LIN {X 0,Y 573.073,Z 538.954,A -85,B 0,C 180,E1 -2243.185,E2 -2243.185} C_VEL
LIN {X 0,Y 573.07,Z 545.679,A -85,B 0,C 180,E1 -2244.369,E2 -2244.369} C_VEL
LIN {X 0,Y 573.028,Z 550.371,A -85,B 0,C 180,E1 -2245.427,E2 -2245.427} C_VEL
LIN {X 0,Y 573.022,Z 553.957,A -85,B 0,C 180,E1 -2246.484,E2 -2246.484} C_VEL
LIN {X 0,Y 572.959,Z 555.808,A -85,B 0,C 180,E1 -2247.187,E2 -2247.187} C_VEL
LIN {X 0,Y 572.939,Z 557.197,A -85,B 0,C 180,E1 -2247.891,E2 -2247.891} C_VEL
LIN {X 0,Y 572.941,Z 558.785,A -85,B 0,C 180,E1 -2249.297,E2 -2249.297} C_VEL
LIN {X 0,Y 572.938,Z 559,A -85,B 0,C 180,E1 -2250,E2 -2250} C_VEL
LIN {X 0,Y 572.946,Z 558.187,A -85,B 0,C 180,E1 -2251.405,E2 -2251.405} C_VEL
LIN {X 0,Y 572.939,Z 557.2,A -85,B 0,C 180,E1 -2252.109,E2 -2252.109} C_VEL
LIN {X 0,Y 572.959,Z 555.811,A -85,B 0,C 180,E1 -2252.812,E2 -2252.812} C_VEL
LIN {X 0,Y 573.014,Z 552.897,A -85,B 0,C 180,E1 -2253.868,E2 -2253.868} C_VEL
LIN {X 0,Y 572.963,Z 548.951,A -85,B 0,C 180,E1 -2254.925,E2 -2254.925} C_VEL
LIN {X 0,Y 573.064,Z 542.879,A -85,B 0,C 180,E1 -2256.16,E2 -2256.16} C_VEL
LIN {X 0,Y 573.119,Z 536.24,A -85,B 0,C 180,E1 -2257.22,E2 -2257.22} C_VEL
LIN {X 0,Y 573.2,Z 527.995,A -85,B 0,C 180,E1 -2258.283,E2 -2258.283} C_VEL
LIN {X 0,Y 573.286,Z 519.544,A -85,B 0,C 180,E1 -2259.17,E2 -2259.17} C_VEL
LIN {X 0,Y 573.43,Z 509.105,A -85,B 0,C 180,E1 -2260.058,E2 -2260.058} C_VEL
LIN {X 0,Y 573.549,Z 497.36,A -85,B 0,C 180,E1 -2260.857,E2 -2260.857} C_VEL
LIN {X 0,Y 573.652,Z 486.295,A -85,B 0,C 180,E1 -2261.447,E2 -2261.447} C_VEL
LIN {X 0,Y 573.758,Z 473.188,A -85,B 0,C 180,E1 -2261.973,E2 -2261.973} C_VEL
LIN {X 0,Y 573.831,Z 460.542,A -85,B 0,C 180,E1 -2262.331,E2 -2262.331} C_VEL
LIN {X 0,Y 573.923,Z 447.356,A -85,B 0,C 180,E1 -2262.553,E2 -2262.553} C_VEL
LIN {X 0,Y 574.016,Z 348.98,A -85,B 0,C 180,E1 -2263.79,E2 -2263.79} C_VEL
LIN {X 0,Y 573.511,Z 345.166,A -85,B 0,C 180,E1 -2263.87,E2 -2263.87} C_VEL
LIN {X 0,Y 573.751,Z 319.651,A -85,B 0,C 180,E1 -2266.729,E2 -2266.729} C_VEL
LIN {X 0,Y 574.013,Z 295.575,A -85,B 0,C 180,E1 -2269.479,E2 -2269.479} C_VEL
LIN {X 0,Y 574.248,Z 274.356,A -85,B 0,C 180,E1 -2271.917,E2 -2271.917} C_VEL
LIN {X 0,Y 574.374,Z 250.622,A -85,B 0,C 180,E1 -2274.583,E2 -2274.583} C_VEL
LIN {X 0,Y 574.422,Z 240.449,A -85,B 0,C 180,E1 -2275.742,E2 -2275.742} C_VEL
LIN {X 0,Y 573.225,Z 234.224,A -85,B 0,C 180,E1 -2276.525,E2 -2276.525} C_VEL
LIN {X 0,Y 573.208,Z 234.087,A -85,B 0,C 180,E1 -2279.368,E2 -2279.368} C_VEL
LIN {X 0,Y 573.223,Z 234.078,A -85,B 0,C 180,E1 -2282.223,E2 -2282.223} C_VEL
LIN {X 0,Y 573.207,Z 234.08,A -85,B 0,C 180,E1 -2284.767,E2 -2284.767} C_VEL
LIN {X 0,Y 573.181,Z 234.084,A -85,B 0,C 180,E1 -2287.81,E2 -2287.81} C_VEL
LIN {X 0,Y 573.201,Z 234.079,A -85,B 0,C 180,E1 -2290.527,E2 -2290.527} C_VEL
LIN {X 0,Y 573.184,Z 234.09,A -85,B 0,C 180,E1 -2293.363,E2 -2293.363} C_VEL
LIN {X 0,Y 573.192,Z 234.08,A -85,B 0,C 180,E1 -2296.335,E2 -2296.335} C_VEL
LIN {X 0,Y 573.236,Z 234.08,A -85,B 0,C 180,E1 -2299.474,E2 -2299.474} C_VEL
LIN {X 0,Y 573.203,Z 234.078,A -85,B 0,C 180,E1 -2302.19,E2 -2302.19} C_VEL
LIN {X 0,Y 573.21,Z 234.085,A -85,B 0,C 180,E1 -2305.23,E2 -2305.23} C_VEL
LIN {X 0,Y 573.205,Z 234.078,A -85,B 0,C 180,E1 -2308.182,E2 -2308.182} C_VEL
LIN {X 0,Y 573.212,Z 234.082,A -85,B 0,C 180,E1 -2310.631,E2 -2310.631} C_VEL
LIN {X 0,Y 573.188,Z 234.082,A -85,B 0,C 180,E1 -2313.514,E2 -2313.514} C_VEL
LIN {X 0,Y 573.178,Z 234.082,A -85,B 0,C 180,E1 -2316.132,E2 -2316.132} C_VEL
LIN {X 0,Y 573.22,Z 234.084,A -85,B 0,C 180,E1 -2318.713,E2 -2318.713} C_VEL
LIN {X 0,Y 573.18,Z 234.083,A -85,B 0,C 180,E1 -2321.41,E2 -2321.41} C_VEL
LIN {X 0,Y 573.2,Z 234.079,A -85,B 0,C 180,E1 -2323.62,E2 -2323.62} C_VEL
LIN {X 0,Y 573.211,Z 234.078,A -85,B 0,C 180,E1 -2325.806,E2 -2325.806} C_VEL
LIN {X 0,Y 573.248,Z 234.082,A -85,B 0,C 180,E1 -2328.745,E2 -2328.745} C_VEL
LIN {X 0,Y 573.214,Z 234.077,A -85,B 0,C 180,E1 -2331.54,E2 -2331.54} C_VEL
LIN {X 0,Y 573.258,Z 234.078,A -85,B 0,C 180,E1 -2334.372,E2 -2334.372} C_VEL
LIN {X 0,Y 573.265,Z 234.072,A -85,B 0,C 180,E1 -2337.189,E2 -2337.189} C_VEL
LIN {X 0,Y 573.283,Z 234.071,A -85,B 0,C 180,E1 -2340,E2 -2340} C_VEL
LIN {X 0,Y 573.276,Z 234.074,A -85,B 0,C 180,E1 -2342.811,E2 -2342.811} C_VEL
LIN {X 0,Y 573.242,Z 234.074,A -85,B 0,C 180,E1 -2345.629,E2 -2345.629} C_VEL
LIN {X 0,Y 573.22,Z 234.085,A -85,B 0,C 180,E1 -2348.461,E2 -2348.461} C_VEL
LIN {X 0,Y 573.22,Z 234.076,A -85,B 0,C 180,E1 -2351.313,E2 -2351.313} C_VEL
LIN {X 0,Y 573.249,Z 234.08,A -85,B 0,C 180,E1 -2354.417,E2 -2354.417} C_VEL
LIN {X 0,Y 573.203,Z 234.079,A -85,B 0,C 180,E1 -2357.114,E2 -2357.114} C_VEL
LIN {X 0,Y 573.215,Z 234.086,A -85,B 0,C 180,E1 -2360.078,E2 -2360.078} C_VEL
LIN {X 0,Y 573.223,Z 234.076,A -85,B 0,C 180,E1 -2363.1,E2 -2363.1} C_VEL
LIN {X 0,Y 573.2,Z 234.081,A -85,B 0,C 180,E1 -2364.386,E2 -2364.386} C_VEL
LIN {X 0,Y 572.558,Z 234.162,A -85,B 0,C 180,E1 -2364.973,E2 -2364.973} C_VEL
LIN {X 0,Y 569.714,Z 234.521,A -85,B 0,C 180,E1 -2365.924,E2 -2365.924} C_VEL
LIN {X 0,Y 567.285,Z 234.819,A -85,B 0,C 180,E1 -2366.69,E2 -2366.69} C_VEL
LIN {X 0,Y 566.226,Z 234.948,A -85,B 0,C 180,E1 -2367.281,E2 -2367.281} C_VEL
LIN {X 0,Y 566.133,Z 234.96,A -85,B 0,C 180,E1 -2367.481,E2 -2367.481} C_VEL
LIN {X 0,Y 566.154,Z 234.958,A -85,B 0,C 180,E1 -2370.595,E2 -2370.595} C_VEL
LIN {X 0,Y 566.151,Z 234.957,A -85,B 0,C 180,E1 -2373.107,E2 -2373.107} C_VEL
LIN {X 0,Y 566.127,Z 234.966,A -85,B 0,C 180,E1 -2375.695,E2 -2375.695} C_VEL
LIN {X 0,Y 566.177,Z 234.955,A -85,B 0,C 180,E1 -2378.556,E2 -2378.556} C_VEL
LIN {X 0,Y 566.127,Z 234.961,A -85,B 0,C 180,E1 -2381.144,E2 -2381.144} C_VEL
LIN {X 0,Y 566.137,Z 234.964,A -85,B 0,C 180,E1 -2384.042,E2 -2384.042} C_VEL
LIN {X 0,Y 566.176,Z 234.955,A -85,B 0,C 180,E1 -2387.086,E2 -2387.086} C_VEL
LIN {X 0,Y 566.178,Z 234.955,A -85,B 0,C 180,E1 -2390.32,E2 -2390.32} C_VEL
LIN {X 0,Y 566.179,Z 234.954,A -85,B 0,C 180,E1 -2392.603,E2 -2392.603} C_VEL
LIN {X 0,Y 566.169,Z 234.958,A -85,B 0,C 180,E1 -2395.181,E2 -2395.181} C_VEL
LIN {X 0,Y 566.209,Z 234.957,A -85,B 0,C 180,E1 -2397.743,E2 -2397.743} C_VEL
LIN {X 0,Y 566.148,Z 234.96,A -85,B 0,C 180,E1 -2401.045,E2 -2401.045} C_VEL
LIN {X 0,Y 566.166,Z 234.965,A -85,B 0,C 180,E1 -2403.457,E2 -2403.457} C_VEL
LIN {X 0,Y 566.15,Z 234.957,A -85,B 0,C 180,E1 -2406.595,E2 -2406.595} C_VEL
LIN {X 0,Y 566.19,Z 234.955,A -85,B 0,C 180,E1 -2408.902,E2 -2408.902} C_VEL
LIN {X 0,Y 566.167,Z 234.962,A -85,B 0,C 180,E1 -2411.172,E2 -2411.172} C_VEL
LIN {X 0,Y 566.163,Z 234.964,A -85,B 0,C 180,E1 -2413.412,E2 -2413.412} C_VEL
LIN {X 0,Y 566.156,Z 234.956,A -85,B 0,C 180,E1 -2416.358,E2 -2416.358} C_VEL
LIN {X 0,Y 566.216,Z 234.958,A -85,B 0,C 180,E1 -2419.27,E2 -2419.27} C_VEL
LIN {X 0,Y 566.172,Z 234.958,A -85,B 0,C 180,E1 -2422.153,E2 -2422.153} C_VEL
LIN {X 0,Y 566.215,Z 235.144,A -85,B 0,C 180,E1 -2424.168,E2 -2424.168} C_VEL
LIN {X 0,Y 566.455,Z 236.257,A -85,B 0,C 180,E1 -2424.282,E2 -2424.282} C_VEL
LIN {X 0,Y 567.145,Z 238.419,A -85,B 0,C 180,E1 -2424.333,E2 -2424.333} C_VEL
LIN {X 0,Y 566.959,Z 324.827,A -85,B 0,C 180,E1 -2425.446,E2 -2425.446} C_VEL
LIN {X 0,Y 566.876,Z 337.961,A -85,B 0,C 180,E1 -2425.757,E2 -2425.757} C_VEL
LIN {X 0,Y 566.752,Z 351.118,A -85,B 0,C 180,E1 -2426.223,E2 -2426.223} C_VEL
LIN {X 0,Y 566.582,Z 362.999,A -85,B 0,C 180,E1 -2426.801,E2 -2426.801} C_VEL
LIN {X 0,Y 566.441,Z 374.363,A -85,B 0,C 180,E1 -2427.511,E2 -2427.511} C_VEL
LIN {X 0,Y 566.31,Z 384.618,A -85,B 0,C 180,E1 -2428.311,E2 -2428.311} C_VEL
LIN {X 0,Y 566.199,Z 393.038,A -85,B 0,C 180,E1 -2429.111,E2 -2429.111} C_VEL
LIN {X 0,Y 566.093,Z 402.198,A -85,B 0,C 180,E1 -2430.178,E2 -2430.178} C_VEL
LIN {X 0,Y 566.004,Z 409.581,A -85,B 0,C 180,E1 -2431.245,E2 -2431.245} C_VEL
LIN {X 0,Y 565.957,Z 416.415,A -85,B 0,C 180,E1 -2432.491,E2 -2432.491} C_VEL
LIN {X 0,Y 565.953,Z 420.936,A -85,B 0,C 180,E1 -2433.56,E2 -2433.56} C_VEL
LIN {X 0,Y 565.937,Z 423.327,A -85,B 0,C 180,E1 -2434.273,E2 -2434.273} C_VEL
LIN {X 0,Y 565.854,Z 425.295,A -85,B 0,C 180,E1 -2434.988,E2 -2434.988} C_VEL
LIN {X 0,Y 565.905,Z 426.843,A -85,B 0,C 180,E1 -2435.702,E2 -2435.702} C_VEL
LIN {X 0,Y 565.921,Z 428.087,A -85,B 0,C 180,E1 -2436.534,E2 -2436.534} C_VEL
LIN {X 0,Y 565.879,Z 428.964,A -85,B 0,C 180,E1 -2437.852,E2 -2437.852} C_VEL
LIN {X 0,Y 565.853,Z 428.888,A -85,B 0,C 180,E1 -2438.572,E2 -2438.572} C_VEL
LIN {X 0,Y 565.829,Z 428.378,A -85,B 0,C 180,E1 -2439.292,E2 -2439.292} C_VEL
LIN {X 0,Y 565.883,Z 427.458,A -85,B 0,C 180,E1 -2440.013,E2 -2440.013} C_VEL
LIN {X 0,Y 565.905,Z 425.164,A -85,B 0,C 180,E1 -2441.153,E2 -2441.153} C_VEL
LIN {X 0,Y 565.926,Z 422.132,A -85,B 0,C 180,E1 -2442.188,E2 -2442.188} C_VEL
LIN {X 0,Y 565.938,Z 417.851,A -85,B 0,C 180,E1 -2443.282,E2 -2443.282} C_VEL
LIN {X 0,Y 565.966,Z 412.226,A -85,B 0,C 180,E1 -2444.398,E2 -2444.398} C_VEL
LIN {X 0,Y 566.052,Z 405.369,A -85,B 0,C 180,E1 -2445.482,E2 -2445.482} C_VEL
LIN {X 0,Y 566.145,Z 398.22,A -85,B 0,C 180,E1 -2446.404,E2 -2446.404} C_VEL
LIN {X 0,Y 566.271,Z 388.548,A -85,B 0,C 180,E1 -2447.422,E2 -2447.422} C_VEL
LIN {X 0,Y 566.386,Z 377.497,A -85,B 0,C 180,E1 -2448.353,E2 -2448.353} C_VEL
LIN {X 0,Y 566.562,Z 366.716,A -85,B 0,C 180,E1 -2449.077,E2 -2449.077} C_VEL
LIN {X 0,Y 566.696,Z 354.767,A -85,B 0,C 180,E1 -2449.704,E2 -2449.704} C_VEL
LIN {X 0,Y 566.847,Z 341.702,A -85,B 0,C 180,E1 -2450.219,E2 -2450.219} C_VEL
LIN {X 0,Y 566.948,Z 329.752,A -85,B 0,C 180,E1 -2450.546,E2 -2450.546} C_VEL
LIN {X 0,Y 566.981,Z 315.181,A -85,B 0,C 180,E1 -2450.782,E2 -2450.782} C_VEL
LIN {X 0,Y 567.039,Z 237.986,A -85,B 0,C 180,E1 -2451.765,E2 -2451.765} C_VEL
LIN {X 0,Y 566.316,Z 235.664,A -85,B 0,C 180,E1 -2451.847,E2 -2451.847} C_VEL
LIN {X 0,Y 566.185,Z 234.985,A -85,B 0,C 180,E1 -2452.006,E2 -2452.006} C_VEL
LIN {X 0,Y 566.181,Z 234.962,A -85,B 0,C 180,E1 -2455.021,E2 -2455.021} C_VEL
LIN {X 0,Y 566.167,Z 234.959,A -85,B 0,C 180,E1 -2457.341,E2 -2457.341} C_VEL
LIN {X 0,Y 566.17,Z 234.955,A -85,B 0,C 180,E1 -2459.77,E2 -2459.77} C_VEL
LIN {X 0,Y 566.202,Z 234.953,A -85,B 0,C 180,E1 -2462.429,E2 -2462.429} C_VEL
LIN {X 0,Y 566.17,Z 234.957,A -85,B 0,C 180,E1 -2464.987,E2 -2464.987} C_VEL
LIN {X 0,Y 566.184,Z 234.95,A -85,B 0,C 180,E1 -2467.461,E2 -2467.461} C_VEL
LIN {X 0,Y 566.204,Z 234.955,A -85,B 0,C 180,E1 -2470.199,E2 -2470.199} C_VEL
LIN {X 0,Y 566.185,Z 234.956,A -85,B 0,C 180,E1 -2473.055,E2 -2473.055} C_VEL
LIN {X 0,Y 566.153,Z 234.96,A -85,B 0,C 180,E1 -2476.053,E2 -2476.053} C_VEL
LIN {X 0,Y 566.198,Z 234.952,A -85,B 0,C 180,E1 -2479.214,E2 -2479.214} C_VEL
LIN {X 0,Y 566.171,Z 234.954,A -85,B 0,C 180,E1 -2481.635,E2 -2481.635} C_VEL
LIN {X 0,Y 566.138,Z 234.966,A -85,B 0,C 180,E1 -2484.306,E2 -2484.306} C_VEL
LIN {X 0,Y 566.204,Z 234.952,A -85,B 0,C 180,E1 -2486.896,E2 -2486.896} C_VEL
LIN {X 0,Y 566.169,Z 234.951,A -85,B 0,C 180,E1 -2489.406,E2 -2489.406} C_VEL
LIN {X 0,Y 566.164,Z 234.958,A -85,B 0,C 180,E1 -2491.854,E2 -2491.854} C_VEL
LIN {X 0,Y 566.231,Z 234.947,A -85,B 0,C 180,E1 -2495.038,E2 -2495.038} C_VEL
LIN {X 0,Y 566.178,Z 234.956,A -85,B 0,C 180,E1 -2498.136,E2 -2498.136} C_VEL
LIN {X 0,Y 566.223,Z 234.949,A -85,B 0,C 180,E1 -2500.613,E2 -2500.613} C_VEL
LIN {X 0,Y 566.169,Z 234.957,A -85,B 0,C 180,E1 -2503.411,E2 -2503.411} C_VEL
LIN {X 0,Y 566.172,Z 234.958,A -85,B 0,C 180,E1 -2506.358,E2 -2506.358} C_VEL
LIN {X 0,Y 566.222,Z 234.95,A -85,B 0,C 180,E1 -2509.27,E2 -2509.27} C_VEL
LIN {X 0,Y 566.18,Z 234.958,A -85,B 0,C 180,E1 -2512.152,E2 -2512.152} C_VEL
LIN {X 0,Y 566.256,Z 234.944,A -85,B 0,C 180,E1 -2515.016,E2 -2515.016} C_VEL
LIN {X 0,Y 566.259,Z 234.951,A -85,B 0,C 180,E1 -2517.866,E2 -2517.866} C_VEL
LIN {X 0,Y 566.267,Z 234.947,A -85,B 0,C 180,E1 -2520,E2 -2520} C_VEL
LIN {X 0,Y 566.241,Z 234.945,A -85,B 0,C 180,E1 -2522.846,E2 -2522.846} C_VEL
LIN {X 0,Y 566.231,Z 234.954,A -85,B 0,C 180,E1 -2525.698,E2 -2525.698} C_VEL
LIN {X 0,Y 566.178,Z 234.953,A -85,B 0,C 180,E1 -2528.566,E2 -2528.566} C_VEL
LIN {X 0,Y 566.23,Z 234.956,A -85,B 0,C 180,E1 -2531.454,E2 -2531.454} C_VEL
LIN {X 0,Y 566.193,Z 234.952,A -85,B 0,C 180,E1 -2534.494,E2 -2534.494} C_VEL
LIN {X 0,Y 566.177,Z 234.963,A -85,B 0,C 180,E1 -2537.332,E2 -2537.332} C_VEL
LIN {X 0,Y 566.189,Z 234.958,A -85,B 0,C 180,E1 -2539.581,E2 -2539.581} C_VEL
LIN {X 0,Y 566.174,Z 234.955,A -85,B 0,C 180,E1 -2541.863,E2 -2541.863} C_VEL
LIN {X 0,Y 566.17,Z 234.962,A -85,B 0,C 180,E1 -2545.021,E2 -2545.021} C_VEL
LIN {X 0,Y 566.154,Z 234.961,A -85,B 0,C 180,E1 -2547.342,E2 -2547.342} C_VEL
LIN {X 0,Y 566.15,Z 234.959,A -85,B 0,C 180,E1 -2549.772,E2 -2549.772} C_VEL
LIN {X 0,Y 566.183,Z 234.954,A -85,B 0,C 180,E1 -2552.428,E2 -2552.428} C_VEL
LIN {X 0,Y 566.158,Z 234.964,A -85,B 0,C 180,E1 -2554.988,E2 -2554.988} C_VEL
LIN {X 0,Y 566.178,Z 234.956,A -85,B 0,C 180,E1 -2557.462,E2 -2557.462} C_VEL
LIN {X 0,Y 566.199,Z 234.952,A -85,B 0,C 180,E1 -2560.2,E2 -2560.2} C_VEL
LIN {X 0,Y 566.141,Z 234.964,A -85,B 0,C 180,E1 -2563.06,E2 -2563.06} C_VEL
LIN {X 0,Y 566.14,Z 234.959,A -85,B 0,C 180,E1 -2566.055,E2 -2566.055} C_VEL
LIN {X 0,Y 566.141,Z 234.965,A -85,B 0,C 180,E1 -2568.858,E2 -2568.858} C_VEL
LIN {X 0,Y 566.153,Z 234.957,A -85,B 0,C 180,E1 -2571.45,E2 -2571.45} C_VEL
LIN {X 0,Y 566.151,Z 234.958,A -85,B 0,C 180,E1 -2573.793,E2 -2573.793} C_VEL
LIN {X 0,Y 566.193,Z 234.957,A -85,B 0,C 180,E1 -2576.269,E2 -2576.269} C_VEL
LIN {X 0,Y 566.166,Z 234.961,A -85,B 0,C 180,E1 -2578.928,E2 -2578.928} C_VEL
LIN {X 0,Y 566.134,Z 234.964,A -85,B 0,C 180,E1 -2581.854,E2 -2581.854} C_VEL
LIN {X 0,Y 566.18,Z 235.187,A -85,B 0,C 180,E1 -2583.372,E2 -2583.372} C_VEL
LIN {X 0,Y 567.401,Z 241.103,A -85,B 0,C 180,E1 -2584.112,E2 -2584.112} C_VEL
LIN {X 0,Y 567.362,Z 259.698,A -85,B 0,C 180,E1 -2586.243,E2 -2586.243} C_VEL
LIN {X 0,Y 567.226,Z 283.598,A -85,B 0,C 180,E1 -2588.942,E2 -2588.942} C_VEL
LIN {X 0,Y 566.989,Z 303.539,A -85,B 0,C 180,E1 -2591.199,E2 -2591.199} C_VEL
LIN {X 0,Y 566.733,Z 326.088,A -85,B 0,C 180,E1 -2593.798,E2 -2593.798} C_VEL
LIN {X 0,Y 566.548,Z 345.155,A -85,B 0,C 180,E1 -2595.956,E2 -2595.956} C_VEL
LIN {X 0,Y 567.173,Z 350.721,A -85,B 0,C 180,E1 -2596.063,E2 -2596.063} C_VEL
LIN {X 0,Y 566.975,Z 454.945,A -85,B 0,C 180,E1 -2597.403,E2 -2597.403} C_VEL
LIN {X 0,Y 566.867,Z 468.217,A -85,B 0,C 180,E1 -2597.719,E2 -2597.719} C_VEL
LIN {X 0,Y 566.728,Z 481.153,A -85,B 0,C 180,E1 -2598.179,E2 -2598.179} C_VEL
LIN {X 0,Y 566.604,Z 493.246,A -85,B 0,C 180,E1 -2598.77,E2 -2598.77} C_VEL
LIN {X 0,Y 566.425,Z 505.483,A -85,B 0,C 180,E1 -2599.545,E2 -2599.545} C_VEL
LIN {X 0,Y 566.297,Z 515.646,A -85,B 0,C 180,E1 -2600.355,E2 -2600.355} C_VEL
LIN {X 0,Y 566.166,Z 524.785,A -85,B 0,C 180,E1 -2601.253,E2 -2601.253} C_VEL
LIN {X 0,Y 566.081,Z 533.688,A -85,B 0,C 180,E1 -2602.33,E2 -2602.33} C_VEL
LIN {X 0,Y 565.967,Z 540.955,A -85,B 0,C 180,E1 -2603.422,E2 -2603.422} C_VEL
LIN {X 0,Y 566.004,Z 545.679,A -85,B 0,C 180,E1 -2604.299,E2 -2604.299} C_VEL
LIN {X 0,Y 565.933,Z 550.372,A -85,B 0,C 180,E1 -2605.37,E2 -2605.37} C_VEL
LIN {X 0,Y 565.927,Z 553.957,A -85,B 0,C 180,E1 -2606.44,E2 -2606.44} C_VEL
LIN {X 0,Y 565.878,Z 555.807,A -85,B 0,C 180,E1 -2607.152,E2 -2607.152} C_VEL
LIN {X 0,Y 565.846,Z 558.184,A -85,B 0,C 180,E1 -2608.576,E2 -2608.576} C_VEL
LIN {X 0,Y 565.839,Z 559,A -85,B 0,C 180,E1 -2610,E2 -2610} C_VEL
LIN {X 0,Y 565.846,Z 558.186,A -85,B 0,C 180,E1 -2611.423,E2 -2611.423} C_VEL
LIN {X 0,Y 565.878,Z 555.811,A -85,B 0,C 180,E1 -2612.847,E2 -2612.847} C_VEL
LIN {X 0,Y 565.926,Z 552.897,A -85,B 0,C 180,E1 -2613.916,E2 -2613.916} C_VEL
LIN {X 0,Y 565.878,Z 548.95,A -85,B 0,C 180,E1 -2614.987,E2 -2614.987} C_VEL
LIN {X 0,Y 566.002,Z 543.869,A -85,B 0,C 180,E1 -2616.058,E2 -2616.058} C_VEL
LIN {X 0,Y 566.039,Z 537.471,A -85,B 0,C 180,E1 -2617.132,E2 -2617.132} C_VEL
LIN {X 0,Y 566.133,Z 529.482,A -85,B 0,C 180,E1 -2618.207,E2 -2618.207} C_VEL
LIN {X 0,Y 566.228,Z 521.34,A -85,B 0,C 180,E1 -2619.105,E2 -2619.105} C_VEL
LIN {X 0,Y 566.35,Z 511.406,A -85,B 0,C 180,E1 -2620.004,E2 -2620.004} C_VEL
LIN {X 0,Y 566.525,Z 500.294,A -85,B 0,C 180,E1 -2620.807,E2 -2620.807} C_VEL
LIN {X 0,Y 566.659,Z 489.186,A -85,B 0,C 180,E1 -2621.445,E2 -2621.445} C_VEL
LIN {X 0,Y 566.741,Z 476.996,A -85,B 0,C 180,E1 -2621.988,E2 -2621.988} C_VEL
LIN {X 0,Y 566.886,Z 464.199,A -85,B 0,C 180,E1 -2622.393,E2 -2622.393} C_VEL
LIN {X 0,Y 566.964,Z 450.64,A -85,B 0,C 180,E1 -2622.664,E2 -2622.664} C_VEL
LIN {X 0,Y 567.122,Z 349.652,A -85,B 0,C 180,E1 -2623.952,E2 -2623.952} C_VEL
LIN {X 0,Y 566.559,Z 345.174,A -85,B 0,C 180,E1 -2624.043,E2 -2624.043} C_VEL
LIN {X 0,Y 566.814,Z 319.831,A -85,B 0,C 180,E1 -2626.919,E2 -2626.919} C_VEL
LIN {X 0,Y 567.118,Z 295.582,A -85,B 0,C 180,E1 -2629.717,E2 -2629.717} C_VEL
LIN {X 0,Y 567.331,Z 270.088,A -85,B 0,C 180,E1 -2632.582,E2 -2632.582} C_VEL
LIN {X 0,Y 567.506,Z 243.009,A -85,B 0,C 180,E1 -2635.685,E2 -2635.685} C_VEL
LIN {X 0,Y 566.731,Z 237.816,A -85,B 0,C 180,E1 -2636.316,E2 -2636.316} C_VEL
LIN {X 0,Y 566.178,Z 235.079,A -85,B 0,C 180,E1 -2636.689,E2 -2636.689} C_VEL
LIN {X 0,Y 566.141,Z 234.966,A -85,B 0,C 180,E1 -2639.771,E2 -2639.771} C_VEL
LIN {X 0,Y 566.171,Z 234.956,A -85,B 0,C 180,E1 -2642.424,E2 -2642.424} C_VEL
LIN {X 0,Y 566.152,Z 234.961,A -85,B 0,C 180,E1 -2644.985,E2 -2644.985} C_VEL
LIN {X 0,Y 566.17,Z 234.963,A -85,B 0,C 180,E1 -2647.462,E2 -2647.462} C_VEL
LIN {X 0,Y 566.154,Z 234.957,A -85,B 0,C 180,E1 -2650.202,E2 -2650.202} C_VEL
LIN {X 0,Y 566.135,Z 234.965,A -85,B 0,C 180,E1 -2653.059,E2 -2653.059} C_VEL
LIN {X 0,Y 566.143,Z 234.958,A -85,B 0,C 180,E1 -2656.053,E2 -2656.053} C_VEL
LIN {X 0,Y 566.162,Z 234.965,A -85,B 0,C 180,E1 -2659.218,E2 -2659.218} C_VEL
LIN {X 0,Y 566.16,Z 234.959,A -85,B 0,C 180,E1 -2661.635,E2 -2661.635} C_VEL
LIN {X 0,Y 566.126,Z 234.961,A -85,B 0,C 180,E1 -2664.305,E2 -2664.305} C_VEL
LIN {X 0,Y 566.149,Z 234.965,A -85,B 0,C 180,E1 -2666.893,E2 -2666.893} C_VEL
LIN {X 0,Y 566.145,Z 234.962,A -85,B 0,C 180,E1 -2669.405,E2 -2669.405} C_VEL
LIN {X 0,Y 566.134,Z 234.959,A -85,B 0,C 180,E1 -2671.853,E2 -2671.853} C_VEL
LIN {X 0,Y 566.161,Z 234.957,A -85,B 0,C 180,E1 -2674.248,E2 -2674.248} C_VEL
LIN {X 0,Y 566.144,Z 234.961,A -85,B 0,C 180,E1 -2677.367,E2 -2677.367} C_VEL
LIN {X 0,Y 566.155,Z 234.957,A -85,B 0,C 180,E1 -2679.661,E2 -2679.661} C_VEL
LIN {X 0,Y 566.154,Z 234.957,A -85,B 0,C 180,E1 -2681.92,E2 -2681.92} C_VEL
LIN {X 0,Y 566.165,Z 234.963,A -85,B 0,C 180,E1 -2684.89,E2 -2684.89} C_VEL
LIN {X 0,Y 566.16,Z 234.956,A -85,B 0,C 180,E1 -2687.817,E2 -2687.817} C_VEL
LIN {X 0,Y 566.136,Z 234.96,A -85,B 0,C 180,E1 -2689.992,E2 -2689.992} C_VEL
LIN {X 0,Y 566.195,Z 234.958,A -85,B 0,C 180,E1 -2692.87,E2 -2692.87} C_VEL
LIN {X 0,Y 566.24,Z 234.949,A -85,B 0,C 180,E1 -2695.016,E2 -2695.016} C_VEL
LIN {X 0,Y 566.242,Z 234.947,A -85,B 0,C 180,E1 -2697.866,E2 -2697.866} C_VEL
LIN {X 0,Y 566.283,Z 234.947,A -85,B 0,C 180,E1 -2700.711,E2 -2700.711} C_VEL
LIN {X 0,Y 566.24,Z 234.95,A -85,B 0,C 180,E1 -2702.846,E2 -2702.846} C_VEL
LIN {X 0,Y 566.212,Z 234.95,A -85,B 0,C 180,E1 -2705.699,E2 -2705.699} C_VEL
LIN {X 0,Y 566.173,Z 234.961,A -85,B 0,C 180,E1 -2708.567,E2 -2708.567} C_VEL
LIN {X 0,Y 566.178,Z 234.954,A -85,B 0,C 180,E1 -2711.456,E2 -2711.456} C_VEL
LIN {X 0,Y 566.204,Z 234.957,A -85,B 0,C 180,E1 -2714.5,E2 -2714.5} C_VEL
LIN {X 0,Y 566.156,Z 234.957,A -85,B 0,C 180,E1 -2717.333,E2 -2717.333} C_VEL
LIN {X 0,Y 566.184,Z 234.955,A -85,B 0,C 180,E1 -2719.582,E2 -2719.582} C_VEL
LIN {X 0,Y 566.169,Z 234.96,A -85,B 0,C 180,E1 -2721.864,E2 -2721.864} C_VEL
LIN {X 0,Y 566.166,Z 234.955,A -85,B 0,C 180,E1 -2725.022,E2 -2725.022} C_VEL
LIN {X 0,Y 566.133,Z 234.96,A -85,B 0,C 180,E1 -2727.481,E2 -2727.481} C_VEL
LIN {X 0,Y 565.447,Z 235.054,A -85,B 0,C 180,E1 -2728.075,E2 -2728.075} C_VEL
LIN {X 0,Y 562.594,Z 235.407,A -85,B 0,C 180,E1 -2729.039,E2 -2729.039} C_VEL
LIN {X 0,Y 560.203,Z 235.705,A -85,B 0,C 180,E1 -2729.815,E2 -2729.815} C_VEL
LIN {X 0,Y 559.189,Z 235.828,A -85,B 0,C 180,E1 -2730.414,E2 -2730.414} C_VEL
LIN {X 0,Y 559.113,Z 235.835,A -85,B 0,C 180,E1 -2730.616,E2 -2730.616} C_VEL
LIN {X 0,Y 559.124,Z 235.833,A -85,B 0,C 180,E1 -2732.718,E2 -2732.718} C_VEL
LIN {X 0,Y 559.103,Z 235.837,A -85,B 0,C 180,E1 -2735.326,E2 -2735.326} C_VEL
LIN {X 0,Y 559.105,Z 235.842,A -85,B 0,C 180,E1 -2738.02,E2 -2738.02} C_VEL
LIN {X 0,Y 559.083,Z 235.838,A -85,B 0,C 180,E1 -2740.819,E2 -2740.819} C_VEL
LIN {X 0,Y 559.084,Z 235.847,A -85,B 0,C 180,E1 -2743.74,E2 -2743.74} C_VEL
LIN {X 0,Y 559.098,Z 235.838,A -85,B 0,C 180,E1 -2746.264,E2 -2746.264} C_VEL
LIN {X 0,Y 559.085,Z 235.84,A -85,B 0,C 180,E1 -2749.183,E2 -2749.183} C_VEL
LIN {X 0,Y 559.115,Z 235.838,A -85,B 0,C 180,E1 -2751.982,E2 -2751.982} C_VEL
LIN {X 0,Y 559.112,Z 235.834,A -85,B 0,C 180,E1 -2754.791,E2 -2754.791} C_VEL
LIN {X 0,Y 559.138,Z 235.837,A -85,B 0,C 180,E1 -2757.368,E2 -2757.368} C_VEL
LIN {X 0,Y 559.099,Z 235.837,A -85,B 0,C 180,E1 -2760.153,E2 -2760.153} C_VEL
LIN {X 0,Y 559.107,Z 235.84,A -85,B 0,C 180,E1 -2763.187,E2 -2763.187} C_VEL
LIN {X 0,Y 559.089,Z 235.846,A -85,B 0,C 180,E1 -2765.493,E2 -2765.493} C_VEL
LIN {X 0,Y 559.131,Z 235.832,A -85,B 0,C 180,E1 -2768.458,E2 -2768.458} C_VEL
LIN {X 0,Y 559.135,Z 235.835,A -85,B 0,C 180,E1 -2770.926,E2 -2770.926} C_VEL
LIN {X 0,Y 559.142,Z 235.838,A -85,B 0,C 180,E1 -2773.197,E2 -2773.197} C_VEL
LIN {X 0,Y 559.135,Z 235.831,A -85,B 0,C 180,E1 -2776.184,E2 -2776.184} C_VEL
LIN {X 0,Y 559.173,Z 235.836,A -85,B 0,C 180,E1 -2779.134,E2 -2779.134} C_VEL
LIN {X 0,Y 559.127,Z 235.836,A -85,B 0,C 180,E1 -2782.053,E2 -2782.053} C_VEL
LIN {X 0,Y 559.174,Z 236.047,A -85,B 0,C 180,E1 -2784.003,E2 -2784.003} C_VEL
LIN {X 0,Y 559.421,Z 237.127,A -85,B 0,C 180,E1 -2784.114,E2 -2784.114} C_VEL
LIN {X 0,Y 560.214,Z 239.499,A -85,B 0,C 180,E1 -2784.173,E2 -2784.173} C_VEL
LIN {X 0,Y 560.037,Z 325.412,A -85,B 0,C 180,E1 -2785.299,E2 -2785.299} C_VEL
LIN {X 0,Y 559.929,Z 339.105,A -85,B 0,C 180,E1 -2785.636,E2 -2785.636} C_VEL
LIN {X 0,Y 559.805,Z 351.403,A -85,B 0,C 180,E1 -2786.086,E2 -2786.086} C_VEL
LIN {X 0,Y 559.611,Z 363.203,A -85,B 0,C 180,E1 -2786.671,E2 -2786.671} C_VEL
LIN {X 0,Y 559.446,Z 374.53,A -85,B 0,C 180,E1 -2787.39,E2 -2787.39} C_VEL
LIN {X 0,Y 559.298,Z 384.759,A -85,B 0,C 180,E1 -2788.2,E2 -2788.2} C_VEL
LIN {X 0,Y 559.137,Z 394.002,A -85,B 0,C 180,E1 -2789.1,E2 -2789.1} C_VEL
LIN {X 0,Y 559.033,Z 402.96,A -85,B 0,C 180,E1 -2790.18,E2 -2790.18} C_VEL
LIN {X 0,Y 558.926,Z 410.21,A -85,B 0,C 180,E1 -2791.261,E2 -2791.261} C_VEL
LIN {X 0,Y 558.855,Z 416.876,A -85,B 0,C 180,E1 -2792.523,E2 -2792.523} C_VEL
LIN {X 0,Y 558.858,Z 421.29,A -85,B 0,C 180,E1 -2793.605,E2 -2793.605} C_VEL
LIN {X 0,Y 558.828,Z 423.63,A -85,B 0,C 180,E1 -2794.328,E2 -2794.328} C_VEL
LIN {X 0,Y 558.769,Z 425.547,A -85,B 0,C 180,E1 -2795.051,E2 -2795.051} C_VEL
LIN {X 0,Y 558.816,Z 427.029,A -85,B 0,C 180,E1 -2795.775,E2 -2795.775} C_VEL
LIN {X 0,Y 558.849,Z 428.109,A -85,B 0,C 180,E1 -2796.536,E2 -2796.536} C_VEL
LIN {X 0,Y 558.797,Z 428.986,A -85,B 0,C 180,E1 -2797.952,E2 -2797.952} C_VEL
LIN {X 0,Y 558.767,Z 428.84,A -85,B 0,C 180,E1 -2798.681,E2 -2798.681} C_VEL
LIN {X 0,Y 558.78,Z 427.295,A -85,B 0,C 180,E1 -2800.142,E2 -2800.142} C_VEL
LIN {X 0,Y 558.807,Z 425.177,A -85,B 0,C 180,E1 -2801.187,E2 -2801.187} C_VEL
LIN {X 0,Y 558.835,Z 421.772,A -85,B 0,C 180,E1 -2802.345,E2 -2802.345} C_VEL
LIN {X 0,Y 558.851,Z 417.383,A -85,B 0,C 180,E1 -2803.453,E2 -2803.453} C_VEL
LIN {X 0,Y 558.914,Z 411.744,A -85,B 0,C 180,E1 -2804.566,E2 -2804.566} C_VEL
LIN {X 0,Y 558.985,Z 404.643,A -85,B 0,C 180,E1 -2805.683,E2 -2805.683} C_VEL
LIN {X 0,Y 559.104,Z 397.338,A -85,B 0,C 180,E1 -2806.617,E2 -2806.617} C_VEL
LIN {X 0,Y 559.273,Z 387.405,A -85,B 0,C 180,E1 -2807.648,E2 -2807.648} C_VEL
LIN {X 0,Y 559.397,Z 377.334,A -85,B 0,C 180,E1 -2808.495,E2 -2808.495} C_VEL
LIN {X 0,Y 559.577,Z 366.85,A -85,B 0,C 180,E1 -2809.208,E2 -2809.208} C_VEL
LIN {X 0,Y 559.723,Z 354.486,A -85,B 0,C 180,E1 -2809.865,E2 -2809.865} C_VEL
LIN {X 0,Y 559.887,Z 342.693,A -85,B 0,C 180,E1 -2810.337,E2 -2810.337} C_VEL
LIN {X 0,Y 560.021,Z 330.255,A -85,B 0,C 180,E1 -2810.692,E2 -2810.692} C_VEL
LIN {X 0,Y 560.058,Z 316.069,A -85,B 0,C 180,E1 -2810.931,E2 -2810.931} C_VEL
LIN {X 0,Y 560.197,Z 239.496,A -85,B 0,C 180,E1 -2811.918,E2 -2811.918} C_VEL
LIN {X 0,Y 559.278,Z 236.553,A -85,B 0,C 180,E1 -2812.014,E2 -2812.014} C_VEL
LIN {X 0,Y 559.153,Z 235.877,A -85,B 0,C 180,E1 -2812.152,E2 -2812.152} C_VEL
LIN {X 0,Y 559.127,Z 235.838,A -85,B 0,C 180,E1 -2815.3,E2 -2815.3} C_VEL
LIN {X 0,Y 559.136,Z 235.835,A -85,B 0,C 180,E1 -2818.374,E2 -2818.374} C_VEL
LIN {X 0,Y 559.142,Z 235.831,A -85,B 0,C 180,E1 -2821.271,E2 -2821.271} C_VEL
LIN {X 0,Y 559.154,Z 235.831,A -85,B 0,C 180,E1 -2823.946,E2 -2823.946} C_VEL
LIN {X 0,Y 559.124,Z 235.832,A -85,B 0,C 180,E1 -2827.109,E2 -2827.109} C_VEL
LIN {X 0,Y 559.155,Z 235.831,A -85,B 0,C 180,E1 -2829.94,E2 -2829.94} C_VEL
LIN {X 0,Y 559.148,Z 235.837,A -85,B 0,C 180,E1 -2832.744,E2 -2832.744} C_VEL
LIN {X 0,Y 559.121,Z 235.834,A -85,B 0,C 180,E1 -2835.763,E2 -2835.763} C_VEL
LIN {X 0,Y 559.12,Z 235.837,A -85,B 0,C 180,E1 -2838.225,E2 -2838.225} C_VEL
LIN {X 0,Y 559.165,Z 235.826,A -85,B 0,C 180,E1 -2841.192,E2 -2841.192} C_VEL
LIN {X 0,Y 559.111,Z 235.834,A -85,B 0,C 180,E1 -2843.787,E2 -2843.787} C_VEL
LIN {X 0,Y 559.154,Z 235.836,A -85,B 0,C 180,E1 -2846.424,E2 -2846.424} C_VEL
LIN {X 0,Y 559.145,Z 235.826,A -85,B 0,C 180,E1 -2848.98,E2 -2848.98} C_VEL
LIN {X 0,Y 559.111,Z 235.834,A -85,B 0,C 180,E1 -2851.628,E2 -2851.628} C_VEL
LIN {X 0,Y 559.155,Z 235.83,A -85,B 0,C 180,E1 -2854.817,E2 -2854.817} C_VEL
LIN {X 0,Y 559.126,Z 235.833,A -85,B 0,C 180,E1 -2857.846,E2 -2857.846} C_VEL
LIN {X 0,Y 559.185,Z 235.827,A -85,B 0,C 180,E1 -2860.494,E2 -2860.494} C_VEL
LIN {X 0,Y 559.147,Z 235.83,A -85,B 0,C 180,E1 -2863.196,E2 -2863.196} C_VEL
LIN {X 0,Y 559.148,Z 235.835,A -85,B 0,C 180,E1 -2866.183,E2 -2866.183} C_VEL
LIN {X 0,Y 559.181,Z 235.826,A -85,B 0,C 180,E1 -2869.133,E2 -2869.133} C_VEL
LIN {X 0,Y 559.133,Z 235.837,A -85,B 0,C 180,E1 -2872.052,E2 -2872.052} C_VEL
LIN {X 0,Y 559.23,Z 235.819,A -85,B 0,C 180,E1 -2874.953,E2 -2874.953} C_VEL
LIN {X 0,Y 559.232,Z 235.827,A -85,B 0,C 180,E1 -2877.839,E2 -2877.839} C_VEL
LIN {X 0,Y 559.237,Z 235.822,A -85,B 0,C 180,E1 -2880,E2 -2880} C_VEL
LIN {X 0,Y 559.21,Z 235.821,A -85,B 0,C 180,E1 -2882.881,E2 -2882.881} C_VEL
LIN {X 0,Y 559.197,Z 235.829,A -85,B 0,C 180,E1 -2885.77,E2 -2885.77} C_VEL
LIN {X 0,Y 559.145,Z 235.829,A -85,B 0,C 180,E1 -2888.675,E2 -2888.675} C_VEL
LIN {X 0,Y 559.187,Z 235.831,A -85,B 0,C 180,E1 -2891.601,E2 -2891.601} C_VEL
LIN {X 0,Y 559.143,Z 235.83,A -85,B 0,C 180,E1 -2894.576,E2 -2894.576} C_VEL
LIN {X 0,Y 559.121,Z 235.838,A -85,B 0,C 180,E1 -2897.558,E2 -2897.558} C_VEL
LIN {X 0,Y 559.152,Z 235.831,A -85,B 0,C 180,E1 -2899.838,E2 -2899.838} C_VEL
LIN {X 0,Y 559.12,Z 235.832,A -85,B 0,C 180,E1 -2902.154,E2 -2902.154} C_VEL
LIN {X 0,Y 559.13,Z 235.841,A -85,B 0,C 180,E1 -2905.178,E2 -2905.178} C_VEL
LIN {X 0,Y 559.098,Z 235.835,A -85,B 0,C 180,E1 -2907.717,E2 -2907.717} C_VEL
LIN {X 0,Y 559.093,Z 235.837,A -85,B 0,C 180,E1 -2910.186,E2 -2910.186} C_VEL
LIN {X 0,Y 559.139,Z 235.835,A -85,B 0,C 180,E1 -2912.716,E2 -2912.716} C_VEL
LIN {X 0,Y 559.108,Z 235.839,A -85,B 0,C 180,E1 -2915.326,E2 -2915.326} C_VEL
LIN {X 0,Y 559.115,Z 235.833,A -85,B 0,C 180,E1 -2918.019,E2 -2918.019} C_VEL
LIN {X 0,Y 559.119,Z 235.842,A -85,B 0,C 180,E1 -2920.816,E2 -2920.816} C_VEL
LIN {X 0,Y 559.093,Z 235.836,A -85,B 0,C 180,E1 -2923.739,E2 -2923.739} C_VEL
LIN {X 0,Y 559.088,Z 235.84,A -85,B 0,C 180,E1 -2926.262,E2 -2926.262} C_VEL
LIN {X 0,Y 559.098,Z 235.837,A -85,B 0,C 180,E1 -2929.183,E2 -2929.183} C_VEL
LIN {X 0,Y 559.094,Z 235.837,A -85,B 0,C 180,E1 -2931.98,E2 -2931.98} C_VEL
LIN {X 0,Y 559.114,Z 235.839,A -85,B 0,C 180,E1 -2934.79,E2 -2934.79} C_VEL
LIN {X 0,Y 559.133,Z 235.832,A -85,B 0,C 180,E1 -2937.368,E2 -2937.368} C_VEL
LIN {X 0,Y 559.093,Z 235.843,A -85,B 0,C 180,E1 -2940.153,E2 -2940.153} C_VEL
LIN {X 0,Y 559.126,Z 235.932,A -85,B 0,C 180,E1 -2943.182,E2 -2943.182} C_VEL
LIN {X 0,Y 560.52,Z 243.305,A -85,B 0,C 180,E1 -2944.133,E2 -2944.133} C_VEL
LIN {X 0,Y 560.376,Z 267.452,A -85,B 0,C 180,E1 -2946.926,E2 -2946.926} C_VEL
LIN {X 0,Y 560.146,Z 292.823,A -85,B 0,C 180,E1 -2949.816,E2 -2949.816} C_VEL
LIN {X 0,Y 559.897,Z 318.228,A -85,B 0,C 180,E1 -2952.681,E2 -2952.681} C_VEL
LIN {X 0,Y 559.589,Z 344.862,A -85,B 0,C 180,E1 -2955.754,E2 -2955.754} C_VEL
LIN {X 0,Y 559.791,Z 347.143,A -85,B 0,C 180,E1 -2955.829,E2 -2955.829} C_VEL
LIN {X 0,Y 560.328,Z 352.509,A -85,B 0,C 180,E1 -2955.912,E2 -2955.912} C_VEL
LIN {X 0,Y 560.058,Z 454.945,A -85,B 0,C 180,E1 -2957.245,E2 -2957.245} C_VEL
LIN {X 0,Y 559.946,Z 468.217,A -85,B 0,C 180,E1 -2957.565,E2 -2957.565} C_VEL
LIN {X 0,Y 559.792,Z 481.155,A -85,B 0,C 180,E1 -2958.031,E2 -2958.031} C_VEL
LIN {X 0,Y 559.634,Z 493.845,A -85,B 0,C 180,E1 -2958.663,E2 -2958.663} C_VEL
LIN {X 0,Y 559.443,Z 505.485,A -85,B 0,C 180,E1 -2959.413,E2 -2959.413} C_VEL
LIN {X 0,Y 559.294,Z 515.646,A -85,B 0,C 180,E1 -2960.233,E2 -2960.233} C_VEL
LIN {X 0,Y 559.134,Z 524.785,A -85,B 0,C 180,E1 -2961.143,E2 -2961.143} C_VEL
LIN {X 0,Y 559.009,Z 533.688,A -85,B 0,C 180,E1 -2962.232,E2 -2962.232} C_VEL
LIN {X 0,Y 558.925,Z 539.739,A -85,B 0,C 180,E1 -2963.14,E2 -2963.14} C_VEL
LIN {X 0,Y 558.935,Z 545.679,A -85,B 0,C 180,E1 -2964.227,E2 -2964.227} C_VEL
LIN {X 0,Y 558.826,Z 550.372,A -85,B 0,C 180,E1 -2965.311,E2 -2965.311} C_VEL
LIN {X 0,Y 558.836,Z 553.957,A -85,B 0,C 180,E1 -2966.395,E2 -2966.395} C_VEL
LIN {X 0,Y 558.799,Z 555.807,A -85,B 0,C 180,E1 -2967.116,E2 -2967.116} C_VEL
LIN {X 0,Y 558.746,Z 558.184,A -85,B 0,C 180,E1 -2968.558,E2 -2968.558} C_VEL
LIN {X 0,Y 558.74,Z 559,A -85,B 0,C 180,E1 -2970,E2 -2970} C_VEL
LIN {X 0,Y 558.746,Z 558.185,A -85,B 0,C 180,E1 -2971.441,E2 -2971.441} C_VEL
LIN {X 0,Y 558.799,Z 555.811,A -85,B 0,C 180,E1 -2972.883,E2 -2972.883} C_VEL
LIN {X 0,Y 558.843,Z 552.897,A -85,B 0,C 180,E1 -2973.966,E2 -2973.966} C_VEL
LIN {X 0,Y 558.798,Z 548.95,A -85,B 0,C 180,E1 -2975.05,E2 -2975.05} C_VEL
LIN {X 0,Y 558.919,Z 543.869,A -85,B 0,C 180,E1 -2976.135,E2 -2976.135} C_VEL
LIN {X 0,Y 558.977,Z 537.471,A -85,B 0,C 180,E1 -2977.222,E2 -2977.222} C_VEL
LIN {X 0,Y 559.098,Z 529.482,A -85,B 0,C 180,E1 -2978.311,E2 -2978.311} C_VEL
LIN {X 0,Y 559.184,Z 521.339,A -85,B 0,C 180,E1 -2979.221,E2 -2979.221} C_VEL
LIN {X 0,Y 559.359,Z 511.405,A -85,B 0,C 180,E1 -2980.131,E2 -2980.131} C_VEL
LIN {X 0,Y 559.53,Z 500.373,A -85,B 0,C 180,E1 -2980.939,E2 -2980.939} C_VEL
LIN {X 0,Y 559.702,Z 488.151,A -85,B 0,C 180,E1 -2981.643,E2 -2981.643} C_VEL
LIN {X 0,Y 559.83,Z 475.784,A -85,B 0,C 180,E1 -2982.184,E2 -2982.184} C_VEL
LIN {X 0,Y 559.983,Z 462.369,A -85,B 0,C 180,E1 -2982.595,E2 -2982.595} C_VEL
LIN {X 0,Y 560.063,Z 449.126,A -85,B 0,C 180,E1 -2982.846,E2 -2982.846} C_VEL
LIN {X 0,Y 560.164,Z 349.774,A -85,B 0,C 180,E1 -2984.127,E2 -2984.127} C_VEL
LIN {X 0,Y 559.579,Z 345.181,A -85,B 0,C 180,E1 -2984.222,E2 -2984.222} C_VEL
LIN {X 0,Y 559.875,Z 320.203,A -85,B 0,C 180,E1 -2987.091,E2 -2987.091} C_VEL
LIN {X 0,Y 560.132,Z 294.543,A -85,B 0,C 180,E1 -2989.992,E2 -2989.992} C_VEL
LIN {X 0,Y 560.367,Z 270.94,A -85,B 0,C 180,E1 -2992.684,E2 -2992.684} C_VEL
LIN {X 0,Y 560.581,Z 244.924,A -85,B 0,C 180,E1 -2995.703,E2 -2995.703} C_VEL
LIN {X 0,Y 560.054,Z 240.406,A -85,B 0,C 180,E1 -2996.253,E2 -2996.253} C_VEL
LIN {X 0,Y 559.122,Z 235.964,A -85,B 0,C 180,E1 -2996.843,E2 -2996.843} C_VEL
LIN {X 0,Y 559.091,Z 235.843,A -85,B 0,C 180,E1 -2999.847,E2 -2999.847} C_VEL
LIN {X 0,Y 559.129,Z 235.834,A -85,B 0,C 180,E1 -3002.716,E2 -3002.716} C_VEL
LIN {X 0,Y 559.105,Z 235.844,A -85,B 0,C 180,E1 -3005.324,E2 -3005.324} C_VEL
LIN {X 0,Y 559.09,Z 235.838,A -85,B 0,C 180,E1 -3008.02,E2 -3008.02} C_VEL
LIN {X 0,Y 559.093,Z 235.839,A -85,B 0,C 180,E1 -3010.816,E2 -3010.816} C_VEL
LIN {X 0,Y 559.084,Z 235.84,A -85,B 0,C 180,E1 -3013.738,E2 -3013.738} C_VEL
LIN {X 0,Y 559.089,Z 235.837,A -85,B 0,C 180,E1 -3016.261,E2 -3016.261} C_VEL
LIN {X 0,Y 559.114,Z 235.844,A -85,B 0,C 180,E1 -3019.184,E2 -3019.184} C_VEL
LIN {X 0,Y 559.11,Z 235.834,A -85,B 0,C 180,E1 -3021.98,E2 -3021.98} C_VEL
LIN {X 0,Y 559.109,Z 235.839,A -85,B 0,C 180,E1 -3024.788,E2 -3024.788} C_VEL
LIN {X 0,Y 559.125,Z 235.837,A -85,B 0,C 180,E1 -3027.367,E2 -3027.367} C_VEL
LIN {X 0,Y 559.093,Z 235.837,A -85,B 0,C 180,E1 -3030.15,E2 -3030.15} C_VEL
LIN {X 0,Y 559.104,Z 235.841,A -85,B 0,C 180,E1 -3033.183,E2 -3033.183} C_VEL
LIN {X 0,Y 559.08,Z 235.84,A -85,B 0,C 180,E1 -3035.491,E2 -3035.491} C_VEL
LIN {X 0,Y 559.128,Z 235.836,A -85,B 0,C 180,E1 -3038.454,E2 -3038.454} C_VEL
LIN {X 0,Y 559.139,Z 235.839,A -85,B 0,C 180,E1 -3040.925,E2 -3040.925} C_VEL
LIN {X 0,Y 559.119,Z 235.833,A -85,B 0,C 180,E1 -3043.947,E2 -3043.947} C_VEL
LIN {X 0,Y 559.123,Z 235.835,A -85,B 0,C 180,E1 -3046.183,E2 -3046.183} C_VEL
LIN {X 0,Y 559.161,Z 235.831,A -85,B 0,C 180,E1 -3049.133,E2 -3049.133} C_VEL
LIN {X 0,Y 559.169,Z 235.829,A -85,B 0,C 180,E1 -3052.053,E2 -3052.053} C_VEL
LIN {X 0,Y 559.216,Z 235.825,A -85,B 0,C 180,E1 -3054.953,E2 -3054.953} C_VEL
LIN {X 0,Y 559.215,Z 235.822,A -85,B 0,C 180,E1 -3057.839,E2 -3057.839} C_VEL
LIN {X 0,Y 559.253,Z 235.822,A -85,B 0,C 180,E1 -3060.72,E2 -3060.72} C_VEL
LIN {X 0,Y 559.205,Z 235.826,A -85,B 0,C 180,E1 -3062.882,E2 -3062.882} C_VEL
LIN {X 0,Y 559.183,Z 235.826,A -85,B 0,C 180,E1 -3065.771,E2 -3065.771} C_VEL
LIN {X 0,Y 559.138,Z 235.836,A -85,B 0,C 180,E1 -3068.675,E2 -3068.675} C_VEL
LIN {X 0,Y 559.141,Z 235.831,A -85,B 0,C 180,E1 -3071.602,E2 -3071.602} C_VEL
LIN {X 0,Y 559.167,Z 235.832,A -85,B 0,C 180,E1 -3074.588,E2 -3074.588} C_VEL
LIN {X 0,Y 559.106,Z 235.836,A -85,B 0,C 180,E1 -3077.559,E2 -3077.559} C_VEL
LIN {X 0,Y 559.146,Z 235.834,A -85,B 0,C 180,E1 -3079.839,E2 -3079.839} C_VEL
LIN {X 0,Y 559.118,Z 235.843,A -85,B 0,C 180,E1 -3082.154,E2 -3082.154} C_VEL
LIN {X 0,Y 559.125,Z 235.832,A -85,B 0,C 180,E1 -3085.178,E2 -3085.178} C_VEL
LIN {X 0,Y 559.087,Z 235.842,A -85,B 0,C 180,E1 -3087.718,E2 -3087.718} C_VEL
LIN {X 0,Y 559.113,Z 235.835,A -85,B 0,C 180,E1 -3090.616,E2 -3090.616} C_VEL
LIN {X 0,Y 558.458,Z 235.916,A -85,B 0,C 180,E1 -3091.218,E2 -3091.218} C_VEL
LIN {X 0,Y 555.595,Z 236.278,A -85,B 0,C 180,E1 -3092.194,E2 -3092.194} C_VEL
LIN {X 0,Y 553.175,Z 236.576,A -85,B 0,C 180,E1 -3092.979,E2 -3092.979} C_VEL
LIN {X 0,Y 552.147,Z 236.706,A -85,B 0,C 180,E1 -3093.586,E2 -3093.586} C_VEL
LIN {X 0,Y 552.071,Z 236.715,A -85,B 0,C 180,E1 -3093.792,E2 -3093.792} C_VEL
LIN {X 0,Y 552.041,Z 236.715,A -85,B 0,C 180,E1 -3096.753,E2 -3096.753} C_VEL
LIN {X 0,Y 552.068,Z 236.716,A -85,B 0,C 180,E1 -3099.533,E2 -3099.533} C_VEL
LIN {X 0,Y 552.071,Z 236.712,A -85,B 0,C 180,E1 -3102.432,E2 -3102.432} C_VEL
LIN {X 0,Y 552.064,Z 236.718,A -85,B 0,C 180,E1 -3105.561,E2 -3105.561} C_VEL
LIN {X 0,Y 552.046,Z 236.714,A -85,B 0,C 180,E1 -3108.549,E2 -3108.549} C_VEL
LIN {X 0,Y 552.088,Z 236.715,A -85,B 0,C 180,E1 -3111.41,E2 -3111.41} C_VEL
LIN {X 0,Y 552.055,Z 236.713,A -85,B 0,C 180,E1 -3114.564,E2 -3114.564} C_VEL
LIN {X 0,Y 552.095,Z 236.712,A -85,B 0,C 180,E1 -3117.158,E2 -3117.158} C_VEL
LIN {X 0,Y 552.067,Z 236.715,A -85,B 0,C 180,E1 -3119.959,E2 -3119.959} C_VEL
LIN {X 0,Y 552.062,Z 236.713,A -85,B 0,C 180,E1 -3122.724,E2 -3122.724} C_VEL
LIN {X 0,Y 552.049,Z 236.719,A -85,B 0,C 180,E1 -3125.159,E2 -3125.159} C_VEL
LIN {X 0,Y 552.048,Z 236.721,A -85,B 0,C 180,E1 -3127.548,E2 -3127.548} C_VEL
LIN {X 0,Y 552.114,Z 236.706,A -85,B 0,C 180,E1 -3130.386,E2 -3130.386} C_VEL
LIN {X 0,Y 552.107,Z 236.711,A -85,B 0,C 180,E1 -3132.976,E2 -3132.976} C_VEL
LIN {X 0,Y 552.095,Z 236.709,A -85,B 0,C 180,E1 -3136.004,E2 -3136.004} C_VEL
LIN {X 0,Y 552.14,Z 236.71,A -85,B 0,C 180,E1 -3138.994,E2 -3138.994} C_VEL
LIN {X 0,Y 552.098,Z 236.713,A -85,B 0,C 180,E1 -3141.951,E2 -3141.951} C_VEL
LIN {X 0,Y 552.128,Z 236.887,A -85,B 0,C 180,E1 -3143.812,E2 -3143.812} C_VEL
LIN {X 0,Y 552.339,Z 237.835,A -85,B 0,C 180,E1 -3143.925,E2 -3143.925} C_VEL
LIN {X 0,Y 553.39,Z 241.159,A -85,B 0,C 180,E1 -3144.009,E2 -3144.009} C_VEL
LIN {X 0,Y 553.147,Z 325.534,A -85,B 0,C 180,E1 -3145.126,E2 -3145.126} C_VEL
LIN {X 0,Y 553.041,Z 338.616,A -85,B 0,C 180,E1 -3145.445,E2 -3145.445} C_VEL
LIN {X 0,Y 552.912,Z 351.136,A -85,B 0,C 180,E1 -3145.9,E2 -3145.9} C_VEL
LIN {X 0,Y 552.697,Z 362.3,A -85,B 0,C 180,E1 -3146.446,E2 -3146.446} C_VEL
LIN {X 0,Y 552.529,Z 373.762,A -85,B 0,C 180,E1 -3147.175,E2 -3147.175} C_VEL
LIN {X 0,Y 552.332,Z 384.057,A -85,B 0,C 180,E1 -3147.995,E2 -3147.995} C_VEL
LIN {X 0,Y 552.137,Z 393.356,A -85,B 0,C 180,E1 -3148.906,E2 -3148.906} C_VEL
LIN {X 0,Y 551.988,Z 402.378,A -85,B 0,C 180,E1 -3150,E2 -3150} C_VEL
LIN {X 0,Y 551.878,Z 409.728,A -85,B 0,C 180,E1 -3151.095,E2 -3151.095} C_VEL
LIN {X 0,Y 551.737,Z 415.651,A -85,B 0,C 180,E1 -3152.19,E2 -3152.19} C_VEL
LIN {X 0,Y 551.781,Z 420.335,A -85,B 0,C 180,E1 -3153.286,E2 -3153.286} C_VEL
LIN {X 0,Y 551.722,Z 423.932,A -85,B 0,C 180,E1 -3154.384,E2 -3154.384} C_VEL
LIN {X 0,Y 551.686,Z 425.793,A -85,B 0,C 180,E1 -3155.116,E2 -3155.116} C_VEL
LIN {X 0,Y 551.732,Z 428.087,A -85,B 0,C 180,E1 -3156.497,E2 -3156.497} C_VEL
LIN {X 0,Y 551.693,Z 428.788,A -85,B 0,C 180,E1 -3157.319,E2 -3157.319} C_VEL
LIN {X 0,Y 551.697,Z 429,A -85,B 0,C 180,E1 -3158.055,E2 -3158.055} C_VEL
LIN {X 0,Y 551.671,Z 428.772,A -85,B 0,C 180,E1 -3158.794,E2 -3158.794} C_VEL
LIN {X 0,Y 551.681,Z 427.133,A -85,B 0,C 180,E1 -3160.274,E2 -3160.274} C_VEL
LIN {X 0,Y 551.72,Z 425.176,A -85,B 0,C 180,E1 -3161.228,E2 -3161.228} C_VEL
LIN {X 0,Y 551.749,Z 421.413,A -85,B 0,C 180,E1 -3162.506,E2 -3162.506} C_VEL
LIN {X 0,Y 551.776,Z 416.916,A -85,B 0,C 180,E1 -3163.629,E2 -3163.629} C_VEL
LIN {X 0,Y 551.851,Z 411.157,A -85,B 0,C 180,E1 -3164.756,E2 -3164.756} C_VEL
LIN {X 0,Y 551.921,Z 403.862,A -85,B 0,C 180,E1 -3165.889,E2 -3165.889} C_VEL
LIN {X 0,Y 552.074,Z 394.775,A -85,B 0,C 180,E1 -3167.025,E2 -3167.025} C_VEL
LIN {X 0,Y 552.29,Z 385.449,A -85,B 0,C 180,E1 -3167.974,E2 -3167.974} C_VEL
LIN {X 0,Y 552.499,Z 374.938,A -85,B 0,C 180,E1 -3168.831,E2 -3168.831} C_VEL
LIN {X 0,Y 552.688,Z 363.903,A -85,B 0,C 180,E1 -3169.55,E2 -3169.55} C_VEL
LIN {X 0,Y 552.853,Z 351.652,A -85,B 0,C 180,E1 -3170.171,E2 -3170.171} C_VEL
LIN {X 0,Y 553.023,Z 338.503,A -85,B 0,C 180,E1 -3170.65,E2 -3170.65} C_VEL
LIN {X 0,Y 553.2,Z 325.717,A -85,B 0,C 180,E1 -3170.959,E2 -3170.959} C_VEL
LIN {X 0,Y 553.342,Z 240.906,A -85,B 0,C 180,E1 -3172.086,E2 -3172.086} C_VEL
LIN {X 0,Y 552.24,Z 237.451,A -85,B 0,C 180,E1 -3172.193,E2 -3172.193} C_VEL
LIN {X 0,Y 552.114,Z 236.771,A -85,B 0,C 180,E1 -3172.321,E2 -3172.321} C_VEL
LIN {X 0,Y 552.084,Z 236.716,A -85,B 0,C 180,E1 -3175.333,E2 -3175.333} C_VEL
LIN {X 0,Y 552.078,Z 236.712,A -85,B 0,C 180,E1 -3178.1,E2 -3178.1} C_VEL
LIN {X 0,Y 552.093,Z 236.712,A -85,B 0,C 180,E1 -3180.609,E2 -3180.609} C_VEL
LIN {X 0,Y 552.106,Z 236.711,A -85,B 0,C 180,E1 -3183.186,E2 -3183.186} C_VEL
LIN {X 0,Y 552.071,Z 236.707,A -85,B 0,C 180,E1 -3185.844,E2 -3185.844} C_VEL
LIN {X 0,Y 552.115,Z 236.71,A -85,B 0,C 180,E1 -3189.06,E2 -3189.06} C_VEL
LIN {X 0,Y 552.069,Z 236.71,A -85,B 0,C 180,E1 -3191.45,E2 -3191.45} C_VEL
LIN {X 0,Y 552.091,Z 236.71,A -85,B 0,C 180,E1 -3193.481,E2 -3193.481} C_VEL
LIN {X 0,Y 552.07,Z 236.716,A -85,B 0,C 180,E1 -3196.572,E2 -3196.572} C_VEL
LIN {X 0,Y 552.105,Z 236.709,A -85,B 0,C 180,E1 -3199.796,E2 -3199.796} C_VEL
LIN {X 0,Y 552.078,Z 236.714,A -85,B 0,C 180,E1 -3202.334,E2 -3202.334} C_VEL
LIN {X 0,Y 552.072,Z 236.713,A -85,B 0,C 180,E1 -3205.05,E2 -3205.05} C_VEL
LIN {X 0,Y 552.107,Z 236.708,A -85,B 0,C 180,E1 -3207.68,E2 -3207.68} C_VEL
LIN {X 0,Y 552.102,Z 236.71,A -85,B 0,C 180,E1 -3210.234,E2 -3210.234} C_VEL
LIN {X 0,Y 552.072,Z 236.712,A -85,B 0,C 180,E1 -3213.012,E2 -3213.012} C_VEL
LIN {X 0,Y 552.097,Z 236.708,A -85,B 0,C 180,E1 -3215.16,E2 -3215.16} C_VEL
LIN {X 0,Y 552.12,Z 236.704,A -85,B 0,C 180,E1 -3218.337,E2 -3218.337} C_VEL
LIN {X 0,Y 552.141,Z 236.702,A -85,B 0,C 180,E1 -3220.674,E2 -3220.674} C_VEL
LIN {X 0,Y 552.084,Z 236.716,A -85,B 0,C 180,E1 -3223.736,E2 -3223.736} C_VEL
LIN {X 0,Y 552.117,Z 236.713,A -85,B 0,C 180,E1 -3226.004,E2 -3226.004} C_VEL
LIN {X 0,Y 552.15,Z 236.701,A -85,B 0,C 180,E1 -3228.993,E2 -3228.993} C_VEL
LIN {X 0,Y 552.102,Z 236.715,A -85,B 0,C 180,E1 -3231.951,E2 -3231.951} C_VEL
LIN {X 0,Y 552.205,Z 236.694,A -85,B 0,C 180,E1 -3234.889,E2 -3234.889} C_VEL
LIN {X 0,Y 552.204,Z 236.703,A -85,B 0,C 180,E1 -3237.812,E2 -3237.812} C_VEL
LIN {X 0,Y 552.206,Z 236.698,A -85,B 0,C 180,E1 -3240,E2 -3240} C_VEL
LIN {X 0,Y 552.179,Z 236.697,A -85,B 0,C 180,E1 -3242.918,E2 -3242.918} C_VEL
LIN {X 0,Y 552.165,Z 236.703,A -85,B 0,C 180,E1 -3245.844,E2 -3245.844} C_VEL
LIN {X 0,Y 552.118,Z 236.705,A -85,B 0,C 180,E1 -3248.786,E2 -3248.786} C_VEL
LIN {X 0,Y 552.142,Z 236.706,A -85,B 0,C 180,E1 -3251.751,E2 -3251.751} C_VEL
LIN {X 0,Y 552.11,Z 236.707,A -85,B 0,C 180,E1 -3254.749,E2 -3254.749} C_VEL
LIN {X 0,Y 552.079,Z 236.712,A -85,B 0,C 180,E1 -3257.789,E2 -3257.789} C_VEL
LIN {X 0,Y 552.113,Z 236.707,A -85,B 0,C 180,E1 -3260.102,E2 -3260.102} C_VEL
LIN {X 0,Y 552.073,Z 236.711,A -85,B 0,C 180,E1 -3262.452,E2 -3262.452} C_VEL
LIN {X 0,Y 552.073,Z 236.717,A -85,B 0,C 180,E1 -3265.334,E2 -3265.334} C_VEL
LIN {X 0,Y 552.046,Z 236.711,A -85,B 0,C 180,E1 -3268.102,E2 -3268.102} C_VEL
LIN {X 0,Y 552.067,Z 236.715,A -85,B 0,C 180,E1 -3270.611,E2 -3270.611} C_VEL
LIN {X 0,Y 552.096,Z 236.712,A -85,B 0,C 180,E1 -3273.187,E2 -3273.187} C_VEL
LIN {X 0,Y 552.061,Z 236.713,A -85,B 0,C 180,E1 -3275.846,E2 -3275.846} C_VEL
LIN {X 0,Y 552.108,Z 236.714,A -85,B 0,C 180,E1 -3279.061,E2 -3279.061} C_VEL
LIN {X 0,Y 552.052,Z 236.716,A -85,B 0,C 180,E1 -3281.452,E2 -3281.452} C_VEL
LIN {X 0,Y 552.066,Z 236.717,A -85,B 0,C 180,E1 -3284.529,E2 -3284.529} C_VEL
LIN {X 0,Y 552.075,Z 236.712,A -85,B 0,C 180,E1 -3287.591,E2 -3287.591} C_VEL
LIN {X 0,Y 552.067,Z 236.716,A -85,B 0,C 180,E1 -3290.468,E2 -3290.468} C_VEL
LIN {X 0,Y 552.047,Z 236.716,A -85,B 0,C 180,E1 -3293.326,E2 -3293.326} C_VEL
LIN {X 0,Y 552.092,Z 236.71,A -85,B 0,C 180,E1 -3295.937,E2 -3295.937} C_VEL
LIN {X 0,Y 552.078,Z 236.717,A -85,B 0,C 180,E1 -3298.538,E2 -3298.538} C_VEL
LIN {X 0,Y 552.067,Z 236.716,A -85,B 0,C 180,E1 -3301.45,E2 -3301.45} C_VEL
LIN {X 0,Y 552.092,Z 236.933,A -85,B 0,C 180,E1 -3303.066,E2 -3303.066} C_VEL
LIN {X 0,Y 553.6,Z 244.763,A -85,B 0,C 180,E1 -3304.066,E2 -3304.066} C_VEL
LIN {X 0,Y 553.397,Z 268.249,A -85,B 0,C 180,E1 -3306.816,E2 -3306.816} C_VEL
LIN {X 0,Y 553.144,Z 293.617,A -85,B 0,C 180,E1 -3309.743,E2 -3309.743} C_VEL
LIN {X 0,Y 552.847,Z 319.773,A -85,B 0,C 180,E1 -3312.726,E2 -3312.726} C_VEL
LIN {X 0,Y 552.614,Z 345.166,A -85,B 0,C 180,E1 -3315.594,E2 -3315.594} C_VEL
LIN {X 0,Y 553.447,Z 352.509,A -85,B 0,C 180,E1 -3315.734,E2 -3315.734} C_VEL
LIN {X 0,Y 553.136,Z 454.945,A -85,B 0,C 180,E1 -3317.083,E2 -3317.083} C_VEL
LIN {X 0,Y 553.028,Z 468.216,A -85,B 0,C 180,E1 -3317.407,E2 -3317.407} C_VEL
LIN {X 0,Y 552.831,Z 481.487,A -85,B 0,C 180,E1 -3317.892,E2 -3317.892} C_VEL
LIN {X 0,Y 552.676,Z 493.742,A -85,B 0,C 180,E1 -3318.512,E2 -3318.512} C_VEL
LIN {X 0,Y 552.469,Z 505.484,A -85,B 0,C 180,E1 -3319.278,E2 -3319.278} C_VEL
LIN {X 0,Y 552.282,Z 515.645,A -85,B 0,C 180,E1 -3320.108,E2 -3320.108} C_VEL
LIN {X 0,Y 552.104,Z 524.785,A -85,B 0,C 180,E1 -3321.029,E2 -3321.029} C_VEL
LIN {X 0,Y 551.96,Z 533.687,A -85,B 0,C 180,E1 -3322.133,E2 -3322.133} C_VEL
LIN {X 0,Y 551.835,Z 540.848,A -85,B 0,C 180,E1 -3323.234,E2 -3323.234} C_VEL
LIN {X 0,Y 551.804,Z 547.365,A -85,B 0,C 180,E1 -3324.518,E2 -3324.518} C_VEL
LIN {X 0,Y 551.764,Z 551.676,A -85,B 0,C 180,E1 -3325.617,E2 -3325.617} C_VEL
LIN {X 0,Y 551.75,Z 553.958,A -85,B 0,C 180,E1 -3326.348,E2 -3326.348} C_VEL
LIN {X 0,Y 551.723,Z 555.807,A -85,B 0,C 180,E1 -3327.079,E2 -3327.079} C_VEL
LIN {X 0,Y 551.645,Z 558.183,A -85,B 0,C 180,E1 -3328.54,E2 -3328.54} C_VEL
LIN {X 0,Y 551.64,Z 559,A -85,B 0,C 180,E1 -3330,E2 -3330} C_VEL
LIN {X 0,Y 551.645,Z 558.185,A -85,B 0,C 180,E1 -3331.46,E2 -3331.46} C_VEL
LIN {X 0,Y 551.723,Z 555.811,A -85,B 0,C 180,E1 -3332.92,E2 -3332.92} C_VEL
LIN {X 0,Y 551.763,Z 552.896,A -85,B 0,C 180,E1 -3334.017,E2 -3334.017} C_VEL
LIN {X 0,Y 551.723,Z 548.95,A -85,B 0,C 180,E1 -3335.115,E2 -3335.115} C_VEL
LIN {X 0,Y 551.814,Z 543.129,A -85,B 0,C 180,E1 -3336.352,E2 -3336.352} C_VEL
LIN {X 0,Y 551.926,Z 536.239,A -85,B 0,C 180,E1 -3337.499,E2 -3337.499} C_VEL
LIN {X 0,Y 552.082,Z 527.996,A -85,B 0,C 180,E1 -3338.602,E2 -3338.602} C_VEL
LIN {X 0,Y 552.222,Z 519.545,A -85,B 0,C 180,E1 -3339.523,E2 -3339.523} C_VEL
LIN {X 0,Y 552.426,Z 509.099,A -85,B 0,C 180,E1 -3340.444,E2 -3340.444} C_VEL
LIN {X 0,Y 552.582,Z 498.136,A -85,B 0,C 180,E1 -3341.224,E2 -3341.224} C_VEL
LIN {X 0,Y 552.781,Z 487.416,A -85,B 0,C 180,E1 -3341.83,E2 -3341.83} C_VEL
LIN {X 0,Y 552.913,Z 475.78,A -85,B 0,C 180,E1 -3342.339,E2 -3342.339} C_VEL
LIN {X 0,Y 553.04,Z 462.368,A -85,B 0,C 180,E1 -3342.755,E2 -3342.755} C_VEL
LIN {X 0,Y 553.163,Z 449.126,A -85,B 0,C 180,E1 -3343.009,E2 -3343.009} C_VEL
LIN {X 0,Y 553.344,Z 350.769,A -85,B 0,C 180,E1 -3344.292,E2 -3344.292} C_VEL
LIN {X 0,Y 552.587,Z 345.189,A -85,B 0,C 180,E1 -3344.406,E2 -3344.406} C_VEL
LIN {X 0,Y 552.863,Z 318.147,A -85,B 0,C 180,E1 -3347.461,E2 -3347.461} C_VEL
LIN {X 0,Y 553.129,Z 291.984,A -85,B 0,C 180,E1 -3350.451,E2 -3350.451} C_VEL
LIN {X 0,Y 553.42,Z 268.419,A -85,B 0,C 180,E1 -3353.183,E2 -3353.183} C_VEL
LIN {X 0,Y 553.631,Z 244.724,A -85,B 0,C 180,E1 -3355.972,E2 -3355.972} C_VEL
LIN {X 0,Y 552.087,Z 236.884,A -85,B 0,C 180,E1 -3356.989,E2 -3356.989} C_VEL
LIN {X 0,Y 552.058,Z 236.72,A -85,B 0,C 180,E1 -3359.767,E2 -3359.767} C_VEL
LIN {X 0,Y 552.09,Z 236.71,A -85,B 0,C 180,E1 -3362.319,E2 -3362.319} C_VEL
LIN {X 0,Y 552.063,Z 236.716,A -85,B 0,C 180,E1 -3364.949,E2 -3364.949} C_VEL
LIN {X 0,Y 552.061,Z 236.715,A -85,B 0,C 180,E1 -3367.881,E2 -3367.881} C_VEL
LIN {X 0,Y 552.06,Z 236.713,A -85,B 0,C 180,E1 -3370.484,E2 -3370.484} C_VEL
LIN {X 0,Y 552.051,Z 236.72,A -85,B 0,C 180,E1 -3373.477,E2 -3373.477} C_VEL
LIN {X 0,Y 552.063,Z 236.713,A -85,B 0,C 180,E1 -3376.572,E2 -3376.572} C_VEL
LIN {X 0,Y 552.091,Z 236.71,A -85,B 0,C 180,E1 -3379.797,E2 -3379.797} C_VEL
LIN {X 0,Y 552.069,Z 236.712,A -85,B 0,C 180,E1 -3382.334,E2 -3382.334} C_VEL
LIN {X 0,Y 552.06,Z 236.722,A -85,B 0,C 180,E1 -3385.049,E2 -3385.049} C_VEL
LIN {X 0,Y 552.083,Z 236.711,A -85,B 0,C 180,E1 -3387.679,E2 -3387.679} C_VEL
LIN {X 0,Y 552.059,Z 236.713,A -85,B 0,C 180,E1 -3390.232,E2 -3390.232} C_VEL
LIN {X 0,Y 552.065,Z 236.721,A -85,B 0,C 180,E1 -3393.012,E2 -3393.012} C_VEL
LIN {X 0,Y 552.055,Z 236.713,A -85,B 0,C 180,E1 -3395.96,E2 -3395.96} C_VEL
LIN {X 0,Y 552.075,Z 236.713,A -85,B 0,C 180,E1 -3398.335,E2 -3398.335} C_VEL
LIN {X 0,Y 552.123,Z 236.712,A -85,B 0,C 180,E1 -3400.673,E2 -3400.673} C_VEL
LIN {X 0,Y 552.067,Z 236.712,A -85,B 0,C 180,E1 -3403.736,E2 -3403.736} C_VEL
LIN {X 0,Y 552.086,Z 236.71,A -85,B 0,C 180,E1 -3406.003,E2 -3406.003} C_VEL
LIN {X 0,Y 552.134,Z 236.708,A -85,B 0,C 180,E1 -3408.993,E2 -3408.993} C_VEL
LIN {X 0,Y 552.124,Z 236.705,A -85,B 0,C 180,E1 -3411.951,E2 -3411.951} C_VEL
LIN {X 0,Y 552.192,Z 236.701,A -85,B 0,C 180,E1 -3414.889,E2 -3414.889} C_VEL
LIN {X 0,Y 552.189,Z 236.697,A -85,B 0,C 180,E1 -3417.812,E2 -3417.812} C_VEL
LIN {X 0,Y 552.223,Z 236.698,A -85,B 0,C 180,E1 -3420.729,E2 -3420.729} C_VEL
LIN {X 0,Y 552.17,Z 236.702,A -85,B 0,C 180,E1 -3422.918,E2 -3422.918} C_VEL
LIN {X 0,Y 552.155,Z 236.703,A -85,B 0,C 180,E1 -3425.845,E2 -3425.845} C_VEL
LIN {X 0,Y 552.11,Z 236.71,A -85,B 0,C 180,E1 -3428.787,E2 -3428.787} C_VEL
LIN {X 0,Y 552.087,Z 236.711,A -85,B 0,C 180,E1 -3431.752,E2 -3431.752} C_VEL
LIN {X 0,Y 552.114,Z 236.708,A -85,B 0,C 180,E1 -3434.749,E2 -3434.749} C_VEL
LIN {X 0,Y 552.067,Z 236.715,A -85,B 0,C 180,E1 -3437.79,E2 -3437.79} C_VEL
LIN {X 0,Y 552.106,Z 236.715,A -85,B 0,C 180,E1 -3440.102,E2 -3440.102} C_VEL
LIN {X 0,Y 552.071,Z 236.716,A -85,B 0,C 180,E1 -3442.452,E2 -3442.452} C_VEL
LIN {X 0,Y 552.066,Z 236.712,A -85,B 0,C 180,E1 -3445.334,E2 -3445.334} C_VEL
LIN {X 0,Y 552.036,Z 236.724,A -85,B 0,C 180,E1 -3448.103,E2 -3448.103} C_VEL
LIN {X 0,Y 552.078,Z 236.712,A -85,B 0,C 180,E1 -3450.612,E2 -3450.612} C_VEL
LIN {X 0,Y 552.084,Z 236.71,A -85,B 0,C 180,E1 -3453.188,E2 -3453.188} C_VEL
LIN {X 0,Y 552.071,Z 236.715,A -85,B 0,C 180,E1 -3453.792,E2 -3453.792} C_VEL
LIN {X 0,Y 551.417,Z 236.801,A -85,B 0,C 180,E1 -3454.4,E2 -3454.4} C_VEL
LIN {X 0,Y 548.546,Z 237.157,A -85,B 0,C 180,E1 -3455.388,E2 -3455.388} C_VEL
LIN {X 0,Y 546.112,Z 237.459,A -85,B 0,C 180,E1 -3456.183,E2 -3456.183} C_VEL
LIN {X 0,Y 545.072,Z 237.583,A -85,B 0,C 180,E1 -3456.798,E2 -3456.798} C_VEL
LIN {X 0,Y 544.99,Z 237.593,A -85,B 0,C 180,E1 -3457.006,E2 -3457.006} C_VEL
LIN {X 0,Y 545.023,Z 237.591,A -85,B 0,C 180,E1 -3459.316,E2 -3459.316} C_VEL
LIN {X 0,Y 545.02,Z 237.594,A -85,B 0,C 180,E1 -3462.109,E2 -3462.109} C_VEL
LIN {X 0,Y 545.01,Z 237.592,A -85,B 0,C 180,E1 -3465.173,E2 -3465.173} C_VEL
LIN {X 0,Y 545.025,Z 237.596,A -85,B 0,C 180,E1 -3467.894,E2 -3467.894} C_VEL
LIN {X 0,Y 545.041,Z 237.587,A -85,B 0,C 180,E1 -3470.816,E2 -3470.816} C_VEL
LIN {X 0,Y 544.999,Z 237.602,A -85,B 0,C 180,E1 -3473.618,E2 -3473.618} C_VEL
LIN {X 0,Y 545.031,Z 237.589,A -85,B 0,C 180,E1 -3476.327,E2 -3476.327} C_VEL
LIN {X 0,Y 545.029,Z 237.59,A -85,B 0,C 180,E1 -3478.951,E2 -3478.951} C_VEL
LIN {X 0,Y 545.035,Z 237.597,A -85,B 0,C 180,E1 -3481.505,E2 -3481.505} C_VEL
LIN {X 0,Y 545.015,Z 237.592,A -85,B 0,C 180,E1 -3483.997,E2 -3483.997} C_VEL
LIN {X 0,Y 545.069,Z 237.583,A -85,B 0,C 180,E1 -3486.441,E2 -3486.441} C_VEL
LIN {X 0,Y 545.041,Z 237.592,A -85,B 0,C 180,E1 -3489.627,E2 -3489.627} C_VEL
LIN {X 0,Y 545.051,Z 237.588,A -85,B 0,C 180,E1 -3492.749,E2 -3492.749} C_VEL
LIN {X 0,Y 545.048,Z 237.588,A -85,B 0,C 180,E1 -3495.819,E2 -3495.819} C_VEL
LIN {X 0,Y 545.088,Z 237.586,A -85,B 0,C 180,E1 -3498.849,E2 -3498.849} C_VEL
LIN {X 0,Y 545.055,Z 237.591,A -85,B 0,C 180,E1 -3501.846,E2 -3501.846} C_VEL
LIN {X 0,Y 545.069,Z 237.755,A -85,B 0,C 180,E1 -3503.622,E2 -3503.622} C_VEL
LIN {X 0,Y 545.309,Z 238.757,A -85,B 0,C 180,E1 -3503.742,E2 -3503.742} C_VEL
LIN {X 0,Y 546.564,Z 243.251,A -85,B 0,C 180,E1 -3503.847,E2 -3503.847} C_VEL
LIN {X 0,Y 546.245,Z 326.929,A -85,B 0,C 180,E1 -3504.972,E2 -3504.972} C_VEL
LIN {X 0,Y 546.146,Z 340.556,A -85,B 0,C 180,E1 -3505.318,E2 -3505.318} C_VEL
LIN {X 0,Y 545.992,Z 353.296,A -85,B 0,C 180,E1 -3505.802,E2 -3505.802} C_VEL
LIN {X 0,Y 545.785,Z 364.874,A -85,B 0,C 180,E1 -3506.401,E2 -3506.401} C_VEL
LIN {X 0,Y 545.55,Z 376.02,A -85,B 0,C 180,E1 -3507.139,E2 -3507.139} C_VEL
LIN {X 0,Y 545.344,Z 386.067,A -85,B 0,C 180,E1 -3507.969,E2 -3507.969} C_VEL
LIN {X 0,Y 545.171,Z 395.106,A -85,B 0,C 180,E1 -3508.892,E2 -3508.892} C_VEL
LIN {X 0,Y 545.003,Z 403.88,A -85,B 0,C 180,E1 -3510,E2 -3510} C_VEL
LIN {X 0,Y 544.831,Z 410.971,A -85,B 0,C 180,E1 -3511.109,E2 -3511.109} C_VEL
LIN {X 0,Y 544.684,Z 416.662,A -85,B 0,C 180,E1 -3512.219,E2 -3512.219} C_VEL
LIN {X 0,Y 544.707,Z 421.128,A -85,B 0,C 180,E1 -3513.329,E2 -3513.329} C_VEL
LIN {X 0,Y 544.641,Z 424.548,A -85,B 0,C 180,E1 -3514.441,E2 -3514.441} C_VEL
LIN {X 0,Y 544.605,Z 426.28,A -85,B 0,C 180,E1 -3515.183,E2 -3515.183} C_VEL
LIN {X 0,Y 544.653,Z 428.505,A -85,B 0,C 180,E1 -3516.669,E2 -3516.669} C_VEL
LIN {X 0,Y 544.606,Z 429.057,A -85,B 0,C 180,E1 -3517.415,E2 -3517.415} C_VEL
LIN {X 0,Y 544.612,Z 429.18,A -85,B 0,C 180,E1 -3518.161,E2 -3518.161} C_VEL
LIN {X 0,Y 544.583,Z 428.261,A -85,B 0,C 180,E1 -3519.658,E2 -3519.658} C_VEL
LIN {X 0,Y 544.589,Z 427.222,A -85,B 0,C 180,E1 -3520.409,E2 -3520.409} C_VEL
LIN {X 0,Y 544.641,Z 425.462,A -85,B 0,C 180,E1 -3521.273,E2 -3521.273} C_VEL
LIN {X 0,Y 544.679,Z 421.45,A -85,B 0,C 180,E1 -3522.671,E2 -3522.671} C_VEL
LIN {X 0,Y 544.748,Z 416.948,A -85,B 0,C 180,E1 -3523.808,E2 -3523.808} C_VEL
LIN {X 0,Y 544.845,Z 411.163,A -85,B 0,C 180,E1 -3524.95,E2 -3524.95} C_VEL
LIN {X 0,Y 544.967,Z 403.854,A -85,B 0,C 180,E1 -3526.097,E2 -3526.097} C_VEL
LIN {X 0,Y 545.156,Z 394.702,A -85,B 0,C 180,E1 -3527.248,E2 -3527.248} C_VEL
LIN {X 0,Y 545.39,Z 385.089,A -85,B 0,C 180,E1 -3528.209,E2 -3528.209} C_VEL
LIN {X 0,Y 545.574,Z 374.306,A -85,B 0,C 180,E1 -3529.079,E2 -3529.079} C_VEL
LIN {X 0,Y 545.82,Z 363.893,A -85,B 0,C 180,E1 -3529.749,E2 -3529.749} C_VEL
LIN {X 0,Y 545.974,Z 352.217,A -85,B 0,C 180,E1 -3530.338,E2 -3530.338} C_VEL
LIN {X 0,Y 546.137,Z 339.75,A -85,B 0,C 180,E1 -3530.799,E2 -3530.799} C_VEL
LIN {X 0,Y 546.295,Z 327.139,A -85,B 0,C 180,E1 -3531.113,E2 -3531.113} C_VEL
LIN {X 0,Y 546.521,Z 259.34,A -85,B 0,C 180,E1 -3532.03,E2 -3532.03} C_VEL
LIN {X 0,Y 546.386,Z 241.924,A -85,B 0,C 180,E1 -3532.266,E2 -3532.266} C_VEL
LIN {X 0,Y 545.238,Z 238.551,A -85,B 0,C 180,E1 -3532.362,E2 -3532.362} C_VEL
LIN {X 0,Y 545.056,Z 237.659,A -85,B 0,C 180,E1 -3532.509,E2 -3532.509} C_VEL
LIN {X 0,Y 545.042,Z 237.595,A -85,B 0,C 180,E1 -3535.183,E2 -3535.183} C_VEL
LIN {X 0,Y 545.044,Z 237.589,A -85,B 0,C 180,E1 -3537.658,E2 -3537.658} C_VEL
LIN {X 0,Y 545.045,Z 237.589,A -85,B 0,C 180,E1 -3540.239,E2 -3540.239} C_VEL
LIN {X 0,Y 545.073,Z 237.589,A -85,B 0,C 180,E1 -3543.06,E2 -3543.06} C_VEL
LIN {X 0,Y 545.021,Z 237.584,A -85,B 0,C 180,E1 -3545.67,E2 -3545.67} C_VEL
LIN {X 0,Y 545.043,Z 237.586,A -85,B 0,C 180,E1 -3548.237,E2 -3548.237} C_VEL
LIN {X 0,Y 545.019,Z 237.591,A -85,B 0,C 180,E1 -3551.12,E2 -3551.12} C_VEL
LIN {X 0,Y 545.037,Z 237.592,A -85,B 0,C 180,E1 -3554.13,E2 -3554.13} C_VEL
LIN {X 0,Y 545.014,Z 237.591,A -85,B 0,C 180,E1 -3556.886,E2 -3556.886} C_VEL
LIN {X 0,Y 545.059,Z 237.587,A -85,B 0,C 180,E1 -3559.856,E2 -3559.856} C_VEL
LIN {X 0,Y 545.013,Z 237.592,A -85,B 0,C 180,E1 -3562.694,E2 -3562.694} C_VEL
LIN {X 0,Y 545.054,Z 237.587,A -85,B 0,C 180,E1 -3565.61,E2 -3565.61} C_VEL
LIN {X 0,Y 545.053,Z 237.588,A -85,B 0,C 180,E1 -3568.321,E2 -3568.321} C_VEL
LIN {X 0,Y 545.054,Z 237.583,A -85,B 0,C 180,E1 -3571.257,E2 -3571.257} C_VEL
LIN {X 0,Y 545.063,Z 237.588,A -85,B 0,C 180,E1 -3574.497,E2 -3574.497} C_VEL
LIN {X 0,Y 545.024,Z 237.583,A -85,B 0,C 180,E1 -3577.241,E2 -3577.241} C_VEL
LIN {X 0,Y 545.108,Z 237.581,A -85,B 0,C 180,E1 -3580.414,E2 -3580.414} C_VEL
LIN {X 0,Y 545.036,Z 237.591,A -85,B 0,C 180,E1 -3583.52,E2 -3583.52} C_VEL
LIN {X 0,Y 545.073,Z 237.589,A -85,B 0,C 180,E1 -3585.819,E2 -3585.819} C_VEL
LIN {X 0,Y 545.107,Z 237.579,A -85,B 0,C 180,E1 -3588.849,E2 -3588.849} C_VEL
LIN {X 0,Y 545.06,Z 237.592,A -85,B 0,C 180,E1 -3591.846,E2 -3591.846} C_VEL
LIN {X 0,Y 545.161,Z 237.571,A -85,B 0,C 180,E1 -3594.822,E2 -3594.822} C_VEL
LIN {X 0,Y 545.176,Z 237.579,A -85,B 0,C 180,E1 -3597.783,E2 -3597.783} C_VEL
LIN {X 0,Y 545.175,Z 237.574,A -85,B 0,C 180,E1 -3600,E2 -3600} C_VEL
LIN {X 0,Y 545.147,Z 237.573,A -85,B 0,C 180,E1 -3602.956,E2 -3602.956} C_VEL
LIN {X 0,Y 545.112,Z 237.581,A -85,B 0,C 180,E1 -3605.92,E2 -3605.92} C_VEL
LIN {X 0,Y 545.079,Z 237.582,A -85,B 0,C 180,E1 -3608.901,E2 -3608.901} C_VEL
LIN {X 0,Y 545.085,Z 237.583,A -85,B 0,C 180,E1 -3611.905,E2 -3611.905} C_VEL
LIN {X 0,Y 545.067,Z 237.586,A -85,B 0,C 180,E1 -3614.944,E2 -3614.944} C_VEL
LIN {X 0,Y 545.045,Z 237.586,A -85,B 0,C 180,E1 -3618.027,E2 -3618.027} C_VEL
LIN {X 0,Y 545.08,Z 237.583,A -85,B 0,C 180,E1 -3620.373,E2 -3620.373} C_VEL
LIN {X 0,Y 545.061,Z 237.589,A -85,B 0,C 180,E1 -3623.56,E2 -3623.56} C_VEL
LIN {X 0,Y 545.03,Z 237.587,A -85,B 0,C 180,E1 -3626.003,E2 -3626.003} C_VEL
LIN {X 0,Y 545.016,Z 237.59,A -85,B 0,C 180,E1 -3628.736,E2 -3628.736} C_VEL
LIN {X 0,Y 545.037,Z 237.589,A -85,B 0,C 180,E1 -3631.677,E2 -3631.677} C_VEL
LIN {X 0,Y 545.039,Z 237.587,A -85,B 0,C 180,E1 -3634.566,E2 -3634.566} C_VEL
LIN {X 0,Y 545.01,Z 237.594,A -85,B 0,C 180,E1 -3637.306,E2 -3637.306} C_VEL
LIN {X 0,Y 545.05,Z 237.586,A -85,B 0,C 180,E1 -3640.144,E2 -3640.144} C_VEL
LIN {X 0,Y 545.011,Z 237.596,A -85,B 0,C 180,E1 -3643.113,E2 -3643.113} C_VEL
LIN {X 0,Y 545.019,Z 237.592,A -85,B 0,C 180,E1 -3646.23,E2 -3646.23} C_VEL
LIN {X 0,Y 545,Z 237.598,A -85,B 0,C 180,E1 -3648.879,E2 -3648.879} C_VEL
LIN {X 0,Y 545.015,Z 237.59,A -85,B 0,C 180,E1 -3651.869,E2 -3651.869} C_VEL
LIN {X 0,Y 545.016,Z 237.595,A -85,B 0,C 180,E1 -3654.531,E2 -3654.531} C_VEL
LIN {X 0,Y 545.048,Z 237.587,A -85,B 0,C 180,E1 -3657.211,E2 -3657.211} C_VEL
LIN {X 0,Y 545.014,Z 237.594,A -85,B 0,C 180,E1 -3659.808,E2 -3659.808} C_VEL
LIN {X 0,Y 545.002,Z 237.621,A -85,B 0,C 180,E1 -3662.773,E2 -3662.773} C_VEL
LIN {X 0,Y 545.082,Z 238.029,A -85,B 0,C 180,E1 -3662.943,E2 -3662.943} C_VEL
LIN {X 0,Y 546.564,Z 245.208,A -85,B 0,C 180,E1 -3663.871,E2 -3663.871} C_VEL
LIN {X 0,Y 546.562,Z 258.862,A -85,B 0,C 180,E1 -3665.501,E2 -3665.501} C_VEL
LIN {X 0,Y 546.265,Z 282.595,A -85,B 0,C 180,E1 -3668.292,E2 -3668.292} C_VEL
LIN {X 0,Y 545.95,Z 306.184,A -85,B 0,C 180,E1 -3671.032,E2 -3671.032} C_VEL
LIN {X 0,Y 545.673,Z 329.635,A -85,B 0,C 180,E1 -3673.732,E2 -3673.732} C_VEL
LIN {X 0,Y 545.555,Z 344.56,A -85,B 0,C 180,E1 -3675.415,E2 -3675.415} C_VEL
LIN {X 0,Y 546.548,Z 354.139,A -85,B 0,C 180,E1 -3675.581,E2 -3675.581} C_VEL
LIN {X 0,Y 546.224,Z 454.552,A -85,B 0,C 180,E1 -3676.917,E2 -3676.917} C_VEL
LIN {X 0,Y 546.064,Z 467.909,A -85,B 0,C 180,E1 -3677.244,E2 -3677.244} C_VEL
LIN {X 0,Y 545.89,Z 481.305,A -85,B 0,C 180,E1 -3677.735,E2 -3677.735} C_VEL
LIN {X 0,Y 545.706,Z 493.316,A -85,B 0,C 180,E1 -3678.341,E2 -3678.341} C_VEL
LIN {X 0,Y 545.503,Z 504.191,A -85,B 0,C 180,E1 -3679.045,E2 -3679.045} C_VEL
LIN {X 0,Y 545.284,Z 514.603,A -85,B 0,C 180,E1 -3679.886,E2 -3679.886} C_VEL
LIN {X 0,Y 545.085,Z 523.112,A -85,B 0,C 180,E1 -3680.725,E2 -3680.725} C_VEL
LIN {X 0,Y 544.978,Z 530.96,A -85,B 0,C 180,E1 -3681.658,E2 -3681.658} C_VEL
LIN {X 0,Y 544.824,Z 538.62,A -85,B 0,C 180,E1 -3682.775,E2 -3682.775} C_VEL
LIN {X 0,Y 544.776,Z 545.678,A -85,B 0,C 180,E1 -3684.076,E2 -3684.076} C_VEL
LIN {X 0,Y 544.628,Z 550.372,A -85,B 0,C 180,E1 -3685.188,E2 -3685.188} C_VEL
LIN {X 0,Y 544.669,Z 553.957,A -85,B 0,C 180,E1 -3686.301,E2 -3686.301} C_VEL
LIN {X 0,Y 544.65,Z 555.806,A -85,B 0,C 180,E1 -3687.041,E2 -3687.041} C_VEL
LIN {X 0,Y 544.546,Z 558.182,A -85,B 0,C 180,E1 -3688.521,E2 -3688.521} C_VEL
LIN {X 0,Y 544.541,Z 559,A -85,B 0,C 180,E1 -3690,E2 -3690} C_VEL
LIN {X 0,Y 544.546,Z 558.184,A -85,B 0,C 180,E1 -3691.479,E2 -3691.479} C_VEL
LIN {X 0,Y 544.65,Z 555.811,A -85,B 0,C 180,E1 -3692.958,E2 -3692.958} C_VEL
LIN {X 0,Y 544.683,Z 552.896,A -85,B 0,C 180,E1 -3694.069,E2 -3694.069} C_VEL
LIN {X 0,Y 544.653,Z 548.95,A -85,B 0,C 180,E1 -3695.182,E2 -3695.182} C_VEL
LIN {X 0,Y 544.728,Z 543.649,A -85,B 0,C 180,E1 -3696.339,E2 -3696.339} C_VEL
LIN {X 0,Y 544.836,Z 537.469,A -85,B 0,C 180,E1 -3697.411,E2 -3697.411} C_VEL
LIN {X 0,Y 545.006,Z 529.481,A -85,B 0,C 180,E1 -3698.528,E2 -3698.528} C_VEL
LIN {X 0,Y 545.152,Z 521.338,A -85,B 0,C 180,E1 -3699.46,E2 -3699.46} C_VEL
LIN {X 0,Y 545.373,Z 511.403,A -85,B 0,C 180,E1 -3700.393,E2 -3700.393} C_VEL
LIN {X 0,Y 545.552,Z 500.54,A -85,B 0,C 180,E1 -3701.211,E2 -3701.211} C_VEL
LIN {X 0,Y 545.766,Z 489.089,A -85,B 0,C 180,E1 -3701.89,E2 -3701.89} C_VEL
LIN {X 0,Y 545.916,Z 476.76,A -85,B 0,C 180,E1 -3702.452,E2 -3702.452} C_VEL
LIN {X 0,Y 546.108,Z 463.863,A -85,B 0,C 180,E1 -3702.873,E2 -3702.873} C_VEL
LIN {X 0,Y 546.232,Z 450.228,A -85,B 0,C 180,E1 -3703.154,E2 -3703.154} C_VEL
LIN {X 0,Y 546.41,Z 351.145,A -85,B 0,C 180,E1 -3704.462,E2 -3704.462} C_VEL
LIN {X 0,Y 545.556,Z 344.489,A -85,B 0,C 180,E1 -3704.59,E2 -3704.59} C_VEL
LIN {X 0,Y 545.826,Z 319.413,A -85,B 0,C 180,E1 -3707.447,E2 -3707.447} C_VEL
LIN {X 0,Y 546.13,Z 292.836,A -85,B 0,C 180,E1 -3710.528,E2 -3710.528} C_VEL
LIN {X 0,Y 546.481,Z 269.284,A -85,B 0,C 180,E1 -3713.294,E2 -3713.294} C_VEL
LIN {X 0,Y 546.761,Z 247.282,A -85,B 0,C 180,E1 -3715.914,E2 -3715.914} C_VEL
LIN {X 0,Y 545.577,Z 240.341,A -85,B 0,C 180,E1 -3716.798,E2 -3716.798} C_VEL
LIN {X 0,Y 545.021,Z 237.681,A -85,B 0,C 180,E1 -3717.194,E2 -3717.194} C_VEL
LIN {X 0,Y 545.012,Z 237.594,A -85,B 0,C 180,E1 -3720.192,E2 -3720.192} C_VEL
LIN {X 0,Y 545.057,Z 237.59,A -85,B 0,C 180,E1 -3723.058,E2 -3723.058} C_VEL
LIN {X 0,Y 545.009,Z 237.596,A -85,B 0,C 180,E1 -3725.669,E2 -3725.669} C_VEL
LIN {X 0,Y 545.012,Z 237.591,A -85,B 0,C 180,E1 -3728.239,E2 -3728.239} C_VEL
LIN {X 0,Y 544.996,Z 237.599,A -85,B 0,C 180,E1 -3731.121,E2 -3731.121} C_VEL
LIN {X 0,Y 545.016,Z 237.59,A -85,B 0,C 180,E1 -3734.132,E2 -3734.132} C_VEL
LIN {X 0,Y 545.007,Z 237.596,A -85,B 0,C 180,E1 -3736.886,E2 -3736.886} C_VEL
LIN {X 0,Y 545.044,Z 237.587,A -85,B 0,C 180,E1 -3739.855,E2 -3739.855} C_VEL
LIN {X 0,Y 545.005,Z 237.595,A -85,B 0,C 180,E1 -3742.693,E2 -3742.693} C_VEL
LIN {X 0,Y 545.037,Z 237.589,A -85,B 0,C 180,E1 -3745.611,E2 -3745.611} C_VEL
LIN {X 0,Y 545.03,Z 237.589,A -85,B 0,C 180,E1 -3748.323,E2 -3748.323} C_VEL
LIN {X 0,Y 545.024,Z 237.591,A -85,B 0,C 180,E1 -3751.503,E2 -3751.503} C_VEL
LIN {X 0,Y 545.009,Z 237.594,A -85,B 0,C 180,E1 -3754.507,E2 -3754.507} C_VEL
LIN {X 0,Y 545.012,Z 237.595,A -85,B 0,C 180,E1 -3757.241,E2 -3757.241} C_VEL
LIN {X 0,Y 545.088,Z 237.584,A -85,B 0,C 180,E1 -3760.414,E2 -3760.414} C_VEL
LIN {X 0,Y 545.019,Z 237.59,A -85,B 0,C 180,E1 -3763.52,E2 -3763.52} C_VEL
LIN {X 0,Y 545.047,Z 237.586,A -85,B 0,C 180,E1 -3765.819,E2 -3765.819} C_VEL
LIN {X 0,Y 545.093,Z 237.587,A -85,B 0,C 180,E1 -3768.849,E2 -3768.849} C_VEL
LIN {X 0,Y 545.073,Z 237.583,A -85,B 0,C 180,E1 -3771.846,E2 -3771.846} C_VEL
LIN {X 0,Y 545.149,Z 237.579,A -85,B 0,C 180,E1 -3774.823,E2 -3774.823} C_VEL
LIN {X 0,Y 545.162,Z 237.572,A -85,B 0,C 180,E1 -3777.784,E2 -3777.784} C_VEL
LIN {X 0,Y 545.193,Z 237.574,A -85,B 0,C 180,E1 -3780.739,E2 -3780.739} C_VEL
LIN {X 0,Y 545.136,Z 237.578,A -85,B 0,C 180,E1 -3782.956,E2 -3782.956} C_VEL
LIN {X 0,Y 545.106,Z 237.581,A -85,B 0,C 180,E1 -3785.92,E2 -3785.92} C_VEL
LIN {X 0,Y 545.053,Z 237.587,A -85,B 0,C 180,E1 -3788.901,E2 -3788.901} C_VEL
LIN {X 0,Y 545.052,Z 237.589,A -85,B 0,C 180,E1 -3791.906,E2 -3791.906} C_VEL
LIN {X 0,Y 545.066,Z 237.585,A -85,B 0,C 180,E1 -3794.944,E2 -3794.944} C_VEL
LIN {X 0,Y 545.036,Z 237.594,A -85,B 0,C 180,E1 -3798.028,E2 -3798.028} C_VEL
LIN {X 0,Y 545.071,Z 237.589,A -85,B 0,C 180,E1 -3800.373,E2 -3800.373} C_VEL
LIN {X 0,Y 545.061,Z 237.586,A -85,B 0,C 180,E1 -3803.561,E2 -3803.561} C_VEL
LIN {X 0,Y 545.021,Z 237.598,A -85,B 0,C 180,E1 -3806.004,E2 -3806.004} C_VEL
LIN {X 0,Y 545.006,Z 237.592,A -85,B 0,C 180,E1 -3808.735,E2 -3808.735} C_VEL
LIN {X 0,Y 545.042,Z 237.587,A -85,B 0,C 180,E1 -3811.05,E2 -3811.05} C_VEL
LIN {X 0,Y 545.027,Z 237.593,A -85,B 0,C 180,E1 -3813.79,E2 -3813.79} C_VEL
LIN {X 0,Y 544.992,Z 237.596,A -85,B 0,C 180,E1 -3816.385,E2 -3816.385} C_VEL
LIN {X 0,Y 544.99,Z 237.593,A -85,B 0,C 180,E1 -3817.006,E2 -3817.006} C_VEL
LIN {X 0,Y 544.331,Z 237.682,A -85,B 0,C 180,E1 -3817.622,E2 -3817.622} C_VEL
LIN {X 0,Y 541.477,Z 238.038,A -85,B 0,C 180,E1 -3818.623,E2 -3818.623} C_VEL
LIN {X 0,Y 539.059,Z 238.339,A -85,B 0,C 180,E1 -3819.43,E2 -3819.43} C_VEL
LIN {X 0,Y 538.019,Z 238.468,A -85,B 0,C 180,E1 -3820.052,E2 -3820.052} C_VEL
LIN {X 0,Y 537.934,Z 238.475,A -85,B 0,C 180,E1 -3820.263,E2 -3820.263} C_VEL
LIN {X 0,Y 537.946,Z 238.471,A -85,B 0,C 180,E1 -3822.98,E2 -3822.98} C_VEL
LIN {X 0,Y 537.993,Z 238.471,A -85,B 0,C 180,E1 -3825.93,E2 -3825.93} C_VEL
LIN {X 0,Y 537.974,Z 238.47,A -85,B 0,C 180,E1 -3828.223,E2 -3828.223} C_VEL
LIN {X 0,Y 537.983,Z 238.469,A -85,B 0,C 180,E1 -3831.168,E2 -3831.168} C_VEL
LIN {X 0,Y 537.953,Z 238.472,A -85,B 0,C 180,E1 -3834.096,E2 -3834.096} C_VEL
LIN {X 0,Y 537.996,Z 238.465,A -85,B 0,C 180,E1 -3836.726,E2 -3836.726} C_VEL
LIN {X 0,Y 537.986,Z 238.475,A -85,B 0,C 180,E1 -3839.565,E2 -3839.565} C_VEL
LIN {X 0,Y 537.972,Z 238.47,A -85,B 0,C 180,E1 -3841.947,E2 -3841.947} C_VEL
LIN {X 0,Y 537.989,Z 238.465,A -85,B 0,C 180,E1 -3844.464,E2 -3844.464} C_VEL
LIN {X 0,Y 537.994,Z 238.467,A -85,B 0,C 180,E1 -3846.928,E2 -3846.928} C_VEL
LIN {X 0,Y 538.037,Z 238.46,A -85,B 0,C 180,E1 -3850.147,E2 -3850.147} C_VEL
LIN {X 0,Y 537.983,Z 238.476,A -85,B 0,C 180,E1 -3853.298,E2 -3853.298} C_VEL
LIN {X 0,Y 538.021,Z 238.465,A -85,B 0,C 180,E1 -3855.63,E2 -3855.63} C_VEL
LIN {X 0,Y 538.039,Z 238.463,A -85,B 0,C 180,E1 -3858.701,E2 -3858.701} C_VEL
LIN {X 0,Y 538.024,Z 238.468,A -85,B 0,C 180,E1 -3861.739,E2 -3861.739} C_VEL
LIN {X 0,Y 538.045,Z 238.57,A -85,B 0,C 180,E1 -3863.41,E2 -3863.41} C_VEL
LIN {X 0,Y 538.225,Z 239.575,A -85,B 0,C 180,E1 -3863.547,E2 -3863.547} C_VEL
LIN {X 0,Y 539.716,Z 244.155,A -85,B 0,C 180,E1 -3863.664,E2 -3863.664} C_VEL
LIN {X 0,Y 539.376,Z 327.181,A -85,B 0,C 180,E1 -3864.791,E2 -3864.791} C_VEL
LIN {X 0,Y 539.269,Z 340.261,A -85,B 0,C 180,E1 -3865.118,E2 -3865.118} C_VEL
LIN {X 0,Y 539.112,Z 353.335,A -85,B 0,C 180,E1 -3865.608,E2 -3865.608} C_VEL
LIN {X 0,Y 538.918,Z 364.342,A -85,B 0,C 180,E1 -3866.168,E2 -3866.168} C_VEL
LIN {X 0,Y 538.704,Z 375.729,A -85,B 0,C 180,E1 -3866.916,E2 -3866.916} C_VEL
LIN {X 0,Y 538.457,Z 385.978,A -85,B 0,C 180,E1 -3867.756,E2 -3867.756} C_VEL
LIN {X 0,Y 538.253,Z 395.226,A -85,B 0,C 180,E1 -3868.691,E2 -3868.691} C_VEL
LIN {X 0,Y 538.033,Z 404.139,A -85,B 0,C 180,E1 -3869.813,E2 -3869.813} C_VEL
LIN {X 0,Y 537.878,Z 411.326,A -85,B 0,C 180,E1 -3870.936,E2 -3870.936} C_VEL
LIN {X 0,Y 537.674,Z 417.964,A -85,B 0,C 180,E1 -3872.248,E2 -3872.248} C_VEL
LIN {X 0,Y 537.687,Z 422.324,A -85,B 0,C 180,E1 -3873.372,E2 -3873.372} C_VEL
LIN {X 0,Y 537.617,Z 425.66,A -85,B 0,C 180,E1 -3874.499,E2 -3874.499} C_VEL
LIN {X 0,Y 537.589,Z 428.583,A -85,B 0,C 180,E1 -3876.003,E2 -3876.003} C_VEL
LIN {X 0,Y 537.622,Z 429.459,A -85,B 0,C 180,E1 -3876.757,E2 -3876.757} C_VEL
LIN {X 0,Y 537.556,Z 429.942,A -85,B 0,C 180,E1 -3877.512,E2 -3877.512} C_VEL
LIN {X 0,Y 537.576,Z 430.004,A -85,B 0,C 180,E1 -3878.268,E2 -3878.268} C_VEL
LIN {X 0,Y 537.537,Z 429.001,A -85,B 0,C 180,E1 -3879.786,E2 -3879.786} C_VEL
LIN {X 0,Y 537.556,Z 427.881,A -85,B 0,C 180,E1 -3880.547,E2 -3880.547} C_VEL
LIN {X 0,Y 537.613,Z 426.239,A -85,B 0,C 180,E1 -3881.347,E2 -3881.347} C_VEL
LIN {X 0,Y 537.665,Z 423.192,A -85,B 0,C 180,E1 -3882.455,E2 -3882.455} C_VEL
LIN {X 0,Y 537.687,Z 418.966,A -85,B 0,C 180,E1 -3883.608,E2 -3883.608} C_VEL
LIN {X 0,Y 537.838,Z 412.911,A -85,B 0,C 180,E1 -3884.877,E2 -3884.877} C_VEL
LIN {X 0,Y 537.94,Z 406.632,A -85,B 0,C 180,E1 -3885.924,E2 -3885.924} C_VEL
LIN {X 0,Y 538.143,Z 399.546,A -85,B 0,C 180,E1 -3886.893,E2 -3886.893} C_VEL
LIN {X 0,Y 538.359,Z 390.901,A -85,B 0,C 180,E1 -3887.865,E2 -3887.865} C_VEL
LIN {X 0,Y 538.544,Z 381.306,A -85,B 0,C 180,E1 -3888.745,E2 -3888.745} C_VEL
LIN {X 0,Y 538.77,Z 370.747,A -85,B 0,C 180,E1 -3889.528,E2 -3889.528} C_VEL
LIN {X 0,Y 539.068,Z 358.647,A -85,B 0,C 180,E1 -3890.232,E2 -3890.232} C_VEL
LIN {X 0,Y 539.166,Z 346.701,A -85,B 0,C 180,E1 -3890.756,E2 -3890.756} C_VEL
LIN {X 0,Y 539.324,Z 333.094,A -85,B 0,C 180,E1 -3891.174,E2 -3891.174} C_VEL
LIN {X 0,Y 539.408,Z 319.438,A -85,B 0,C 180,E1 -3891.42,E2 -3891.42} C_VEL
LIN {X 0,Y 539.66,Z 243.663,A -85,B 0,C 180,E1 -3892.435,E2 -3892.435} C_VEL
LIN {X 0,Y 538.176,Z 239.309,A -85,B 0,C 180,E1 -3892.563,E2 -3892.563} C_VEL
LIN {X 0,Y 538.017,Z 238.527,A -85,B 0,C 180,E1 -3892.716,E2 -3892.716} C_VEL
LIN {X 0,Y 537.994,Z 238.469,A -85,B 0,C 180,E1 -3895.66,E2 -3895.66} C_VEL
LIN {X 0,Y 538.004,Z 238.466,A -85,B 0,C 180,E1 -3898.052,E2 -3898.052} C_VEL
LIN {X 0,Y 538.008,Z 238.464,A -85,B 0,C 180,E1 -3900.627,E2 -3900.627} C_VEL
LIN {X 0,Y 538.021,Z 238.465,A -85,B 0,C 180,E1 -3903.278,E2 -3903.278} C_VEL
LIN {X 0,Y 537.988,Z 238.461,A -85,B 0,C 180,E1 -3906.004,E2 -3906.004} C_VEL
LIN {X 0,Y 538.007,Z 238.471,A -85,B 0,C 180,E1 -3908.83,E2 -3908.83} C_VEL
LIN {X 0,Y 537.994,Z 238.464,A -85,B 0,C 180,E1 -3911.874,E2 -3911.874} C_VEL
LIN {X 0,Y 537.992,Z 238.47,A -85,B 0,C 180,E1 -3914.863,E2 -3914.863} C_VEL
LIN {X 0,Y 537.984,Z 238.468,A -85,B 0,C 180,E1 -3918.126,E2 -3918.126} C_VEL
LIN {X 0,Y 538.004,Z 238.462,A -85,B 0,C 180,E1 -3921.168,E2 -3921.168} C_VEL
LIN {X 0,Y 537.96,Z 238.471,A -85,B 0,C 180,E1 -3924.093,E2 -3924.093} C_VEL
LIN {X 0,Y 538.027,Z 238.464,A -85,B 0,C 180,E1 -3926.727,E2 -3926.727} C_VEL
LIN {X 0,Y 538.01,Z 238.457,A -85,B 0,C 180,E1 -3929.558,E2 -3929.558} C_VEL
LIN {X 0,Y 537.988,Z 238.468,A -85,B 0,C 180,E1 -3931.947,E2 -3931.947} C_VEL
LIN {X 0,Y 538.04,Z 238.463,A -85,B 0,C 180,E1 -3934.465,E2 -3934.465} C_VEL
LIN {X 0,Y 538.003,Z 238.458,A -85,B 0,C 180,E1 -3936.927,E2 -3936.927} C_VEL
LIN {X 0,Y 538.074,Z 238.459,A -85,B 0,C 180,E1 -3940.147,E2 -3940.147} C_VEL
LIN {X 0,Y 537.986,Z 238.467,A -85,B 0,C 180,E1 -3943.298,E2 -3943.298} C_VEL
LIN {X 0,Y 538.042,Z 238.462,A -85,B 0,C 180,E1 -3945.63,E2 -3945.63} C_VEL
LIN {X 0,Y 538.067,Z 238.456,A -85,B 0,C 180,E1 -3948.701,E2 -3948.701} C_VEL
LIN {X 0,Y 538.031,Z 238.465,A -85,B 0,C 180,E1 -3951.739,E2 -3951.739} C_VEL
LIN {X 0,Y 538.12,Z 238.449,A -85,B 0,C 180,E1 -3954.754,E2 -3954.754} C_VEL
LIN {X 0,Y 538.149,Z 238.454,A -85,B 0,C 180,E1 -3957.754,E2 -3957.754} C_VEL
LIN {X 0,Y 538.145,Z 238.449,A -85,B 0,C 180,E1 -3960,E2 -3960} C_VEL
LIN {X 0,Y 538.115,Z 238.449,A -85,B 0,C 180,E1 -3962.994,E2 -3962.994} C_VEL
LIN {X 0,Y 538.064,Z 238.458,A -85,B 0,C 180,E1 -3965.998,E2 -3965.998} C_VEL
LIN {X 0,Y 538.033,Z 238.461,A -85,B 0,C 180,E1 -3969.018,E2 -3969.018} C_VEL
LIN {X 0,Y 538.044,Z 238.458,A -85,B 0,C 180,E1 -3972.063,E2 -3972.063} C_VEL
LIN {X 0,Y 538.029,Z 238.466,A -85,B 0,C 180,E1 -3975.144,E2 -3975.144} C_VEL
LIN {X 0,Y 537.998,Z 238.463,A -85,B 0,C 180,E1 -3978.271,E2 -3978.271} C_VEL
LIN {X 0,Y 538.024,Z 238.463,A -85,B 0,C 180,E1 -3980.652,E2 -3980.652} C_VEL
LIN {X 0,Y 537.998,Z 238.466,A -85,B 0,C 180,E1 -3983.878,E2 -3983.878} C_VEL
LIN {X 0,Y 537.974,Z 238.466,A -85,B 0,C 180,E1 -3986.37,E2 -3986.37} C_VEL
LIN {X 0,Y 537.985,Z 238.468,A -85,B 0,C 180,E1 -3988.926,E2 -3988.926} C_VEL
LIN {X 0,Y 537.991,Z 238.465,A -85,B 0,C 180,E1 -3991.885,E2 -3991.885} C_VEL
LIN {X 0,Y 537.989,Z 238.465,A -85,B 0,C 180,E1 -3994.615,E2 -3994.615} C_VEL
LIN {X 0,Y 537.974,Z 238.467,A -85,B 0,C 180,E1 -3997.879,E2 -3997.879} C_VEL
LIN {X 0,Y 537.992,Z 238.473,A -85,B 0,C 180,E1 -4000.781,E2 -4000.781} C_VEL
LIN {X 0,Y 537.993,Z 238.465,A -85,B 0,C 180,E1 -4004.071,E2 -4004.071} C_VEL
LIN {X 0,Y 537.949,Z 238.477,A -85,B 0,C 180,E1 -4007.021,E2 -4007.021} C_VEL
LIN {X 0,Y 537.985,Z 238.466,A -85,B 0,C 180,E1 -4009.261,E2 -4009.261} C_VEL
LIN {X 0,Y 537.96,Z 238.47,A -85,B 0,C 180,E1 -4012.12,E2 -4012.12} C_VEL
LIN {X 0,Y 537.991,Z 238.466,A -85,B 0,C 180,E1 -4015.386,E2 -4015.386} C_VEL
LIN {X 0,Y 537.992,Z 238.468,A -85,B 0,C 180,E1 -4018.116,E2 -4018.116} C_VEL
LIN {X 0,Y 537.983,Z 238.473,A -85,B 0,C 180,E1 -4021.096,E2 -4021.096} C_VEL
LIN {X 0,Y 538.009,Z 238.721,A -85,B 0,C 180,E1 -4022.746,E2 -4022.746} C_VEL
LIN {X 0,Y 539.742,Z 247.936,A -85,B 0,C 180,E1 -4023.956,E2 -4023.956} C_VEL
LIN {X 0,Y 539.475,Z 271.548,A -85,B 0,C 180,E1 -4026.792,E2 -4026.792} C_VEL
LIN {X 0,Y 539.082,Z 298.115,A -85,B 0,C 180,E1 -4029.933,E2 -4029.933} C_VEL
LIN {X 0,Y 538.751,Z 323.742,A -85,B 0,C 180,E1 -4032.932,E2 -4032.932} C_VEL
LIN {X 0,Y 538.494,Z 343.756,A -85,B 0,C 180,E1 -4035.223,E2 -4035.223} C_VEL
LIN {X 0,Y 539.664,Z 353.984,A -85,B 0,C 180,E1 -4035.403,E2 -4035.403} C_VEL
LIN {X 0,Y 539.29,Z 453.663,A -85,B 0,C 180,E1 -4036.745,E2 -4036.745} C_VEL
LIN {X 0,Y 539.113,Z 467.025,A -85,B 0,C 180,E1 -4037.076,E2 -4037.076} C_VEL
LIN {X 0,Y 538.9,Z 480.422,A -85,B 0,C 180,E1 -4037.574,E2 -4037.574} C_VEL
LIN {X 0,Y 538.707,Z 492.445,A -85,B 0,C 180,E1 -4038.187,E2 -4038.187} C_VEL
LIN {X 0,Y 538.451,Z 504.736,A -85,B 0,C 180,E1 -4038.995,E2 -4038.995} C_VEL
LIN {X 0,Y 538.208,Z 515.069,A -85,B 0,C 180,E1 -4039.846,E2 -4039.846} C_VEL
LIN {X 0,Y 538.006,Z 524.381,A -85,B 0,C 180,E1 -4040.792,E2 -4040.792} C_VEL
LIN {X 0,Y 537.851,Z 533.471,A -85,B 0,C 180,E1 -4041.925,E2 -4041.925} C_VEL
LIN {X 0,Y 537.708,Z 540.777,A -85,B 0,C 180,E1 -4043.056,E2 -4043.056} C_VEL
LIN {X 0,Y 537.693,Z 545.666,A -85,B 0,C 180,E1 -4043.998,E2 -4043.998} C_VEL
LIN {X 0,Y 537.54,Z 550.372,A -85,B 0,C 180,E1 -4045.125,E2 -4045.125} C_VEL
LIN {X 0,Y 537.591,Z 553.957,A -85,B 0,C 180,E1 -4046.252,E2 -4046.252} C_VEL
LIN {X 0,Y 537.551,Z 555.806,A -85,B 0,C 180,E1 -4047.002,E2 -4047.002} C_VEL
LIN {X 0,Y 537.452,Z 558.181,A -85,B 0,C 180,E1 -4048.501,E2 -4048.501} C_VEL
LIN {X 0,Y 537.442,Z 559,A -85,B 0,C 180,E1 -4050,E2 -4050} C_VEL
LIN {X 0,Y 537.452,Z 558.183,A -85,B 0,C 180,E1 -4051.498,E2 -4051.498} C_VEL
LIN {X 0,Y 537.551,Z 555.811,A -85,B 0,C 180,E1 -4052.997,E2 -4052.997} C_VEL
LIN {X 0,Y 537.603,Z 552.896,A -85,B 0,C 180,E1 -4054.123,E2 -4054.123} C_VEL
LIN {X 0,Y 537.587,Z 548.949,A -85,B 0,C 180,E1 -4055.25,E2 -4055.25} C_VEL
LIN {X 0,Y 537.642,Z 544.102,A -85,B 0,C 180,E1 -4056.325,E2 -4056.325} C_VEL
LIN {X 0,Y 537.771,Z 537.336,A -85,B 0,C 180,E1 -4057.509,E2 -4057.509} C_VEL
LIN {X 0,Y 537.93,Z 529.179,A -85,B 0,C 180,E1 -4058.641,E2 -4058.641} C_VEL
LIN {X 0,Y 538.115,Z 520.879,A -85,B 0,C 180,E1 -4059.585,E2 -4059.585} C_VEL
LIN {X 0,Y 538.337,Z 510.772,A -85,B 0,C 180,E1 -4060.531,E2 -4060.531} C_VEL
LIN {X 0,Y 538.508,Z 500.811,A -85,B 0,C 180,E1 -4061.289,E2 -4061.289} C_VEL
LIN {X 0,Y 538.72,Z 489.79,A -85,B 0,C 180,E1 -4061.964,E2 -4061.964} C_VEL
LIN {X 0,Y 538.911,Z 477.041,A -85,B 0,C 180,E1 -4062.569,E2 -4062.569} C_VEL
LIN {X 0,Y 539.157,Z 463.923,A -85,B 0,C 180,E1 -4063.018,E2 -4063.018} C_VEL
LIN {X 0,Y 539.318,Z 450.872,A -85,B 0,C 180,E1 -4063.301,E2 -4063.301} C_VEL
LIN {X 0,Y 539.57,Z 352.284,A -85,B 0,C 180,E1 -4064.623,E2 -4064.623} C_VEL
LIN {X 0,Y 538.493,Z 343.732,A -85,B 0,C 180,E1 -4064.78,E2 -4064.78} C_VEL
LIN {X 0,Y 538.783,Z 320.46,A -85,B 0,C 180,E1 -4067.458,E2 -4067.458} C_VEL
LIN {X 0,Y 539.141,Z 294.828,A -85,B 0,C 180,E1 -4070.471,E2 -4070.471} C_VEL
LIN {X 0,Y 539.514,Z 270.126,A -85,B 0,C 180,E1 -4073.409,E2 -4073.409} C_VEL
LIN {X 0,Y 539.827,Z 248.148,A -85,B 0,C 180,E1 -4076.063,E2 -4076.063} C_VEL
LIN {X 0,Y 537.982,Z 238.594,A -85,B 0,C 180,E1 -4077.336,E2 -4077.336} C_VEL
LIN {X 0,Y 537.966,Z 238.476,A -85,B 0,C 180,E1 -4079.763,E2 -4079.763} C_VEL
LIN {X 0,Y 537.999,Z 238.466,A -85,B 0,C 180,E1 -4082.383,E2 -4082.383} C_VEL
LIN {X 0,Y 537.977,Z 238.473,A -85,B 0,C 180,E1 -4085.085,E2 -4085.085} C_VEL
LIN {X 0,Y 537.96,Z 238.469,A -85,B 0,C 180,E1 -4088.385,E2 -4088.385} C_VEL
LIN {X 0,Y 537.98,Z 238.469,A -85,B 0,C 180,E1 -4090.781,E2 -4090.781} C_VEL
LIN {X 0,Y 537.987,Z 238.466,A -85,B 0,C 180,E1 -4094.07,E2 -4094.07} C_VEL
LIN {X 0,Y 537.959,Z 238.475,A -85,B 0,C 180,E1 -4097.018,E2 -4097.018} C_VEL
LIN {X 0,Y 537.99,Z 238.465,A -85,B 0,C 180,E1 -4100.2,E2 -4100.2} C_VEL
LIN {X 0,Y 537.959,Z 238.478,A -85,B 0,C 180,E1 -4103.062,E2 -4103.062} C_VEL
LIN {X 0,Y 537.98,Z 238.467,A -85,B 0,C 180,E1 -4105.824,E2 -4105.824} C_VEL
LIN {X 0,Y 537.977,Z 238.469,A -85,B 0,C 180,E1 -4108.496,E2 -4108.496} C_VEL
LIN {X 0,Y 537.971,Z 238.475,A -85,B 0,C 180,E1 -4111.095,E2 -4111.095} C_VEL
LIN {X 0,Y 537.967,Z 238.469,A -85,B 0,C 180,E1 -4113.629,E2 -4113.629} C_VEL
LIN {X 0,Y 537.993,Z 238.465,A -85,B 0,C 180,E1 -4116.122,E2 -4116.122} C_VEL
LIN {X 0,Y 537.995,Z 238.469,A -85,B 0,C 180,E1 -4118.545,E2 -4118.545} C_VEL
LIN {X 0,Y 537.993,Z 238.473,A -85,B 0,C 180,E1 -4120.938,E2 -4120.938} C_VEL
LIN {X 0,Y 537.97,Z 238.47,A -85,B 0,C 180,E1 -4123.297,E2 -4123.297} C_VEL
LIN {X 0,Y 538.021,Z 238.461,A -85,B 0,C 180,E1 -4125.63,E2 -4125.63} C_VEL
LIN {X 0,Y 538.056,Z 238.467,A -85,B 0,C 180,E1 -4128.701,E2 -4128.701} C_VEL
LIN {X 0,Y 538.035,Z 238.46,A -85,B 0,C 180,E1 -4131.739,E2 -4131.739} C_VEL
LIN {X 0,Y 538.108,Z 238.457,A -85,B 0,C 180,E1 -4134.755,E2 -4134.755} C_VEL
LIN {X 0,Y 538.136,Z 238.447,A -85,B 0,C 180,E1 -4137.755,E2 -4137.755} C_VEL
LIN {X 0,Y 538.163,Z 238.449,A -85,B 0,C 180,E1 -4140.748,E2 -4140.748} C_VEL
LIN {X 0,Y 538.101,Z 238.453,A -85,B 0,C 180,E1 -4142.995,E2 -4142.995} C_VEL
LIN {X 0,Y 538.064,Z 238.459,A -85,B 0,C 180,E1 -4145.998,E2 -4145.998} C_VEL
LIN {X 0,Y 538.01,Z 238.464,A -85,B 0,C 180,E1 -4149.019,E2 -4149.019} C_VEL
LIN {X 0,Y 538.023,Z 238.467,A -85,B 0,C 180,E1 -4152.064,E2 -4152.064} C_VEL
LIN {X 0,Y 538.025,Z 238.461,A -85,B 0,C 180,E1 -4155.145,E2 -4155.145} C_VEL
LIN {X 0,Y 537.99,Z 238.474,A -85,B 0,C 180,E1 -4158.272,E2 -4158.272} C_VEL
LIN {X 0,Y 538.015,Z 238.465,A -85,B 0,C 180,E1 -4160.653,E2 -4160.653} C_VEL
LIN {X 0,Y 537.996,Z 238.464,A -85,B 0,C 180,E1 -4163.073,E2 -4163.073} C_VEL
LIN {X 0,Y 537.976,Z 238.47,A -85,B 0,C 180,E1 -4165.661,E2 -4165.661} C_VEL
LIN {X 0,Y 537.959,Z 238.479,A -85,B 0,C 180,E1 -4168.055,E2 -4168.055} C_VEL
LIN {X 0,Y 537.99,Z 238.466,A -85,B 0,C 180,E1 -4170.629,E2 -4170.629} C_VEL
LIN {X 0,Y 538.01,Z 238.464,A -85,B 0,C 180,E1 -4173.28,E2 -4173.28} C_VEL
LIN {X 0,Y 537.945,Z 238.479,A -85,B 0,C 180,E1 -4176.009,E2 -4176.009} C_VEL
LIN {X 0,Y 537.975,Z 238.467,A -85,B 0,C 180,E1 -4178.834,E2 -4178.834} C_VEL
LIN {X 0,Y 537.934,Z 238.475,A -85,B 0,C 180,E1 -4180.263,E2 -4180.263} C_VEL
LIN {X 0,Y 537.269,Z 238.556,A -85,B 0,C 180,E1 -4180.888,E2 -4180.888} C_VEL
LIN {X 0,Y 534.426,Z 238.917,A -85,B 0,C 180,E1 -4181.903,E2 -4181.903} C_VEL
LIN {X 0,Y 532.024,Z 239.218,A -85,B 0,C 180,E1 -4182.721,E2 -4182.721} C_VEL
LIN {X 0,Y 530.994,Z 239.343,A -85,B 0,C 180,E1 -4183.352,E2 -4183.352} C_VEL
LIN {X 0,Y 530.911,Z 239.351,A -85,B 0,C 180,E1 -4183.565,E2 -4183.565} C_VEL
LIN {X 0,Y 530.919,Z 239.347,A -85,B 0,C 180,E1 -4186.502,E2 -4186.502} C_VEL
LIN {X 0,Y 530.908,Z 239.355,A -85,B 0,C 180,E1 -4189.562,E2 -4189.562} C_VEL
LIN {X 0,Y 530.923,Z 239.346,A -85,B 0,C 180,E1 -4192.49,E2 -4192.49} C_VEL
LIN {X 0,Y 530.959,Z 239.346,A -85,B 0,C 180,E1 -4195.309,E2 -4195.309} C_VEL
LIN {X 0,Y 530.951,Z 239.345,A -85,B 0,C 180,E1 -4198.032,E2 -4198.032} C_VEL
LIN {X 0,Y 530.932,Z 239.346,A -85,B 0,C 180,E1 -4200.886,E2 -4200.886} C_VEL
LIN {X 0,Y 530.937,Z 239.35,A -85,B 0,C 180,E1 -4203.254,E2 -4203.254} C_VEL
LIN {X 0,Y 530.952,Z 239.344,A -85,B 0,C 180,E1 -4205.97,E2 -4205.97} C_VEL
LIN {X 0,Y 530.968,Z 239.345,A -85,B 0,C 180,E1 -4209.062,E2 -4209.062} C_VEL
LIN {X 0,Y 530.973,Z 239.339,A -85,B 0,C 180,E1 -4212.277,E2 -4212.277} C_VEL
LIN {X 0,Y 530.976,Z 239.346,A -85,B 0,C 180,E1 -4215.435,E2 -4215.435} C_VEL
LIN {X 0,Y 530.999,Z 239.338,A -85,B 0,C 180,E1 -4218.549,E2 -4218.549} C_VEL
LIN {X 0,Y 530.973,Z 239.347,A -85,B 0,C 180,E1 -4221.629,E2 -4221.629} C_VEL
LIN {X 0,Y 531.03,Z 239.425,A -85,B 0,C 180,E1 -4223.204,E2 -4223.204} C_VEL
LIN {X 0,Y 531.156,Z 240.238,A -85,B 0,C 180,E1 -4223.337,E2 -4223.337} C_VEL
LIN {X 0,Y 532.846,Z 245.529,A -85,B 0,C 180,E1 -4223.482,E2 -4223.482} C_VEL
LIN {X 0,Y 532.507,Z 328.556,A -85,B 0,C 180,E1 -4224.628,E2 -4224.628} C_VEL
LIN {X 0,Y 532.372,Z 342.203,A -85,B 0,C 180,E1 -4224.983,E2 -4224.983} C_VEL
LIN {X 0,Y 532.226,Z 354.426,A -85,B 0,C 180,E1 -4225.456,E2 -4225.456} C_VEL
LIN {X 0,Y 532.017,Z 365.366,A -85,B 0,C 180,E1 -4226.024,E2 -4226.024} C_VEL
LIN {X 0,Y 531.785,Z 376.717,A -85,B 0,C 180,E1 -4226.781,E2 -4226.781} C_VEL
LIN {X 0,Y 531.517,Z 386.94,A -85,B 0,C 180,E1 -4227.632,E2 -4227.632} C_VEL
LIN {X 0,Y 531.32,Z 395.302,A -85,B 0,C 180,E1 -4228.484,E2 -4228.484} C_VEL
LIN {X 0,Y 531.084,Z 403.032,A -85,B 0,C 180,E1 -4229.432,E2 -4229.432} C_VEL
LIN {X 0,Y 530.919,Z 410.6,A -85,B 0,C 180,E1 -4230.569,E2 -4230.569} C_VEL
LIN {X 0,Y 530.689,Z 417.566,A -85,B 0,C 180,E1 -4231.898,E2 -4231.898} C_VEL
LIN {X 0,Y 530.637,Z 422.207,A -85,B 0,C 180,E1 -4233.037,E2 -4233.037} C_VEL
LIN {X 0,Y 530.587,Z 425.776,A -85,B 0,C 180,E1 -4234.178,E2 -4234.178} C_VEL
LIN {X 0,Y 530.56,Z 428.362,A -85,B 0,C 180,E1 -4235.321,E2 -4235.321} C_VEL
LIN {X 0,Y 530.57,Z 430.113,A -85,B 0,C 180,E1 -4236.552,E2 -4236.552} C_VEL
LIN {X 0,Y 530.507,Z 430.811,A -85,B 0,C 180,E1 -4237.613,E2 -4237.613} C_VEL
LIN {X 0,Y 530.488,Z 430.479,A -85,B 0,C 180,E1 -4239.148,E2 -4239.148} C_VEL
LIN {X 0,Y 530.493,Z 429.725,A -85,B 0,C 180,E1 -4239.917,E2 -4239.917} C_VEL
LIN {X 0,Y 530.588,Z 427.015,A -85,B 0,C 180,E1 -4241.424,E2 -4241.424} C_VEL
LIN {X 0,Y 530.643,Z 423.698,A -85,B 0,C 180,E1 -4242.623,E2 -4242.623} C_VEL
LIN {X 0,Y 530.691,Z 419.367,A -85,B 0,C 180,E1 -4243.791,E2 -4243.791} C_VEL
LIN {X 0,Y 530.868,Z 413.588,A -85,B 0,C 180,E1 -4245.001,E2 -4245.001} C_VEL
LIN {X 0,Y 531.002,Z 406.76,A -85,B 0,C 180,E1 -4246.137,E2 -4246.137} C_VEL
LIN {X 0,Y 531.221,Z 397.895,A -85,B 0,C 180,E1 -4247.314,E2 -4247.314} C_VEL
LIN {X 0,Y 531.493,Z 388.659,A -85,B 0,C 180,E1 -4248.303,E2 -4248.303} C_VEL
LIN {X 0,Y 531.726,Z 378.331,A -85,B 0,C 180,E1 -4249.195,E2 -4249.195} C_VEL
LIN {X 0,Y 532.031,Z 366.736,A -85,B 0,C 180,E1 -4249.987,E2 -4249.987} C_VEL
LIN {X 0,Y 532.245,Z 354.726,A -85,B 0,C 180,E1 -4250.624,E2 -4250.624} C_VEL
LIN {X 0,Y 532.378,Z 342.24,A -85,B 0,C 180,E1 -4251.109,E2 -4251.109} C_VEL
LIN {X 0,Y 532.545,Z 330.014,A -85,B 0,C 180,E1 -4251.432,E2 -4251.432} C_VEL
LIN {X 0,Y 532.602,Z 307.86,A -85,B 0,C 180,E1 -4251.763,E2 -4251.763} C_VEL
LIN {X 0,Y 532.733,Z 244.892,A -85,B 0,C 180,E1 -4252.621,E2 -4252.621} C_VEL
LIN {X 0,Y 531.157,Z 240.38,A -85,B 0,C 180,E1 -4252.747,E2 -4252.747} C_VEL
LIN {X 0,Y 530.991,Z 239.473,A -85,B 0,C 180,E1 -4252.88,E2 -4252.88} C_VEL
LIN {X 0,Y 530.964,Z 239.345,A -85,B 0,C 180,E1 -4255.899,E2 -4255.899} C_VEL
LIN {X 0,Y 530.99,Z 239.343,A -85,B 0,C 180,E1 -4259.125,E2 -4259.125} C_VEL
LIN {X 0,Y 530.966,Z 239.338,A -85,B 0,C 180,E1 -4262.099,E2 -4262.099} C_VEL
LIN {X 0,Y 530.959,Z 239.342,A -85,B 0,C 180,E1 -4264.848,E2 -4264.848} C_VEL
LIN {X 0,Y 530.936,Z 239.339,A -85,B 0,C 180,E1 -4267.509,E2 -4267.509} C_VEL
LIN {X 0,Y 530.946,Z 239.351,A -85,B 0,C 180,E1 -4270.435,E2 -4270.435} C_VEL
LIN {X 0,Y 530.936,Z 239.345,A -85,B 0,C 180,E1 -4273.497,E2 -4273.497} C_VEL
LIN {X 0,Y 530.922,Z 239.349,A -85,B 0,C 180,E1 -4276.5,E2 -4276.5} C_VEL
LIN {X 0,Y 530.947,Z 239.344,A -85,B 0,C 180,E1 -4279.563,E2 -4279.563} C_VEL
LIN {X 0,Y 530.928,Z 239.346,A -85,B 0,C 180,E1 -4282.582,E2 -4282.582} C_VEL
LIN {X 0,Y 530.967,Z 239.341,A -85,B 0,C 180,E1 -4285.308,E2 -4285.308} C_VEL
LIN {X 0,Y 530.961,Z 239.346,A -85,B 0,C 180,E1 -4288.031,E2 -4288.031} C_VEL
LIN {X 0,Y 530.983,Z 239.336,A -85,B 0,C 180,E1 -4290.874,E2 -4290.874} C_VEL
LIN {X 0,Y 530.968,Z 239.349,A -85,B 0,C 180,E1 -4294.164,E2 -4294.164} C_VEL
LIN {X 0,Y 530.945,Z 239.338,A -85,B 0,C 180,E1 -4296.602,E2 -4296.602} C_VEL
LIN {X 0,Y 530.99,Z 239.329,A -85,B 0,C 180,E1 -4299.061,E2 -4299.061} C_VEL
LIN {X 0,Y 530.964,Z 239.341,A -85,B 0,C 180,E1 -4301.478,E2 -4301.478} C_VEL
LIN {X 0,Y 530.982,Z 239.337,A -85,B 0,C 180,E1 -4304.65,E2 -4304.65} C_VEL
LIN {X 0,Y 531.016,Z 239.341,A -85,B 0,C 180,E1 -4307.774,E2 -4307.774} C_VEL
LIN {X 0,Y 530.962,Z 239.343,A -85,B 0,C 180,E1 -4310.091,E2 -4310.091} C_VEL
LIN {X 0,Y 531.003,Z 239.337,A -85,B 0,C 180,E1 -4313.159,E2 -4313.159} C_VEL
LIN {X 0,Y 530.974,Z 239.343,A -85,B 0,C 180,E1 -4315.445,E2 -4315.445} C_VEL
LIN {X 0,Y 531.121,Z 239.329,A -85,B 0,C 180,E1 -4317.725,E2 -4317.725} C_VEL
LIN {X 0,Y 531.114,Z 239.325,A -85,B 0,C 180,E1 -4320,E2 -4320} C_VEL
LIN {X 0,Y 531.083,Z 239.325,A -85,B 0,C 180,E1 -4323.034,E2 -4323.034} C_VEL
LIN {X 0,Y 531.023,Z 239.334,A -85,B 0,C 180,E1 -4326.078,E2 -4326.078} C_VEL
LIN {X 0,Y 530.995,Z 239.339,A -85,B 0,C 180,E1 -4329.139,E2 -4329.139} C_VEL
LIN {X 0,Y 531.038,Z 239.335,A -85,B 0,C 180,E1 -4331.669,E2 -4331.669} C_VEL
LIN {X 0,Y 531.01,Z 239.337,A -85,B 0,C 180,E1 -4334.95,E2 -4334.95} C_VEL
LIN {X 0,Y 530.971,Z 239.342,A -85,B 0,C 180,E1 -4337.724,E2 -4337.724} C_VEL
LIN {X 0,Y 531.006,Z 239.336,A -85,B 0,C 180,E1 -4340.128,E2 -4340.128} C_VEL
LIN {X 0,Y 530.932,Z 239.345,A -85,B 0,C 180,E1 -4342.574,E2 -4342.574} C_VEL
LIN {X 0,Y 530.938,Z 239.352,A -85,B 0,C 180,E1 -4345.061,E2 -4345.061} C_VEL
LIN {X 0,Y 530.944,Z 239.341,A -85,B 0,C 180,E1 -4347.599,E2 -4347.599} C_VEL
LIN {X 0,Y 530.926,Z 239.346,A -85,B 0,C 180,E1 -4350.2,E2 -4350.2} C_VEL
LIN {X 0,Y 530.957,Z 239.348,A -85,B 0,C 180,E1 -4352.867,E2 -4352.867} C_VEL
LIN {X 0,Y 530.924,Z 239.347,A -85,B 0,C 180,E1 -4355.622,E2 -4355.622} C_VEL
LIN {X 0,Y 530.953,Z 239.346,A -85,B 0,C 180,E1 -4358.653,E2 -4358.653} C_VEL
LIN {X 0,Y 530.946,Z 239.346,A -85,B 0,C 180,E1 -4361.44,E2 -4361.44} C_VEL
LIN {X 0,Y 530.956,Z 239.347,A -85,B 0,C 180,E1 -4364.55,E2 -4364.55} C_VEL
LIN {X 0,Y 530.901,Z 239.35,A -85,B 0,C 180,E1 -4367.536,E2 -4367.536} C_VEL
LIN {X 0,Y 530.932,Z 239.346,A -85,B 0,C 180,E1 -4370.552,E2 -4370.552} C_VEL
LIN {X 0,Y 530.901,Z 239.351,A -85,B 0,C 180,E1 -4373.438,E2 -4373.438} C_VEL
LIN {X 0,Y 530.947,Z 239.347,A -85,B 0,C 180,E1 -4376.225,E2 -4376.225} C_VEL
LIN {X 0,Y 530.933,Z 239.352,A -85,B 0,C 180,E1 -4378.92,E2 -4378.92} C_VEL
LIN {X 0,Y 530.925,Z 239.351,A -85,B 0,C 180,E1 -4381.541,E2 -4381.541} C_VEL
LIN {X 0,Y 530.964,Z 239.553,A -85,B 0,C 180,E1 -4382.563,E2 -4382.563} C_VEL
LIN {X 0,Y 532.76,Z 248.55,A -85,B 0,C 180,E1 -4383.771,E2 -4383.771} C_VEL
LIN {X 0,Y 532.6,Z 264.087,A -85,B 0,C 180,E1 -4385.675,E2 -4385.675} C_VEL
LIN {X 0,Y 532.31,Z 284.199,A -85,B 0,C 180,E1 -4388.102,E2 -4388.102} C_VEL
LIN {X 0,Y 531.915,Z 307.767,A -85,B 0,C 180,E1 -4390.913,E2 -4390.913} C_VEL
LIN {X 0,Y 531.572,Z 331.203,A -85,B 0,C 180,E1 -4393.683,E2 -4393.683} C_VEL
LIN {X 0,Y 531.453,Z 342.841,A -85,B 0,C 180,E1 -4395.021,E2 -4395.021} C_VEL
LIN {X 0,Y 532.789,Z 355.119,A -85,B 0,C 180,E1 -4395.237,E2 -4395.237} C_VEL
LIN {X 0,Y 532.377,Z 452.776,A -85,B 0,C 180,E1 -4396.57,E2 -4396.57} C_VEL
LIN {X 0,Y 532.18,Z 466.143,A -85,B 0,C 180,E1 -4396.905,E2 -4396.905} C_VEL
LIN {X 0,Y 531.952,Z 478.408,A -85,B 0,C 180,E1 -4397.36,E2 -4397.36} C_VEL
LIN {X 0,Y 531.692,Z 491.081,A -85,B 0,C 180,E1 -4398,E2 -4398} C_VEL
LIN {X 0,Y 531.414,Z 502.543,A -85,B 0,C 180,E1 -4398.751,E2 -4398.751} C_VEL
LIN {X 0,Y 531.172,Z 513.127,A -85,B 0,C 180,E1 -4399.614,E2 -4399.614} C_VEL
LIN {X 0,Y 530.985,Z 521.798,A -85,B 0,C 180,E1 -4400.477,E2 -4400.477} C_VEL
LIN {X 0,Y 530.827,Z 529.811,A -85,B 0,C 180,E1 -4401.434,E2 -4401.434} C_VEL
LIN {X 0,Y 530.674,Z 537.649,A -85,B 0,C 180,E1 -4402.581,E2 -4402.581} C_VEL
LIN {X 0,Y 530.604,Z 544.885,A -85,B 0,C 180,E1 -4403.917,E2 -4403.917} C_VEL
LIN {X 0,Y 530.46,Z 549.693,A -85,B 0,C 180,E1 -4405.059,E2 -4405.059} C_VEL
LIN {X 0,Y 530.516,Z 553.388,A -85,B 0,C 180,E1 -4406.202,E2 -4406.202} C_VEL
LIN {X 0,Y 530.486,Z 555.288,A -85,B 0,C 180,E1 -4406.962,E2 -4406.962} C_VEL
LIN {X 0,Y 530.411,Z 556.707,A -85,B 0,C 180,E1 -4407.722,E2 -4407.722} C_VEL
LIN {X 0,Y 530.355,Z 558.341,A -85,B 0,C 180,E1 -4409.24,E2 -4409.24} C_VEL
LIN {X 0,Y 530.356,Z 558.563,A -85,B 0,C 180,E1 -4410,E2 -4410} C_VEL
LIN {X 0,Y 530.355,Z 558.342,A -85,B 0,C 180,E1 -4410.759,E2 -4410.759} C_VEL
LIN {X 0,Y 530.411,Z 556.713,A -85,B 0,C 180,E1 -4412.278,E2 -4412.278} C_VEL
LIN {X 0,Y 530.486,Z 555.296,A -85,B 0,C 180,E1 -4413.037,E2 -4413.037} C_VEL
LIN {X 0,Y 530.522,Z 552.303,A -85,B 0,C 180,E1 -4414.178,E2 -4414.178} C_VEL
LIN {X 0,Y 530.524,Z 548.247,A -85,B 0,C 180,E1 -4415.32,E2 -4415.32} C_VEL
LIN {X 0,Y 530.594,Z 542.438,A -85,B 0,C 180,E1 -4416.578,E2 -4416.578} C_VEL
LIN {X 0,Y 530.719,Z 535.227,A -85,B 0,C 180,E1 -4417.801,E2 -4417.801} C_VEL
LIN {X 0,Y 530.89,Z 526.811,A -85,B 0,C 180,E1 -4418.948,E2 -4418.948} C_VEL
LIN {X 0,Y 531.08,Z 518.194,A -85,B 0,C 180,E1 -4419.906,E2 -4419.906} C_VEL
LIN {X 0,Y 531.339,Z 507.569,A -85,B 0,C 180,E1 -4420.864,E2 -4420.864} C_VEL
LIN {X 0,Y 531.599,Z 496.486,A -85,B 0,C 180,E1 -4421.67,E2 -4421.67} C_VEL
LIN {X 0,Y 531.807,Z 485.591,A -85,B 0,C 180,E1 -4422.303,E2 -4422.303} C_VEL
LIN {X 0,Y 532.043,Z 473.827,A -85,B 0,C 180,E1 -4422.831,E2 -4422.831} C_VEL
LIN {X 0,Y 532.282,Z 460.31,A -85,B 0,C 180,E1 -4423.262,E2 -4423.262} C_VEL
LIN {X 0,Y 532.444,Z 446.977,A -85,B 0,C 180,E1 -4423.525,E2 -4423.525} C_VEL
LIN {X 0,Y 532.633,Z 352.612,A -85,B 0,C 180,E1 -4424.802,E2 -4424.802} C_VEL
LIN {X 0,Y 531.447,Z 342.922,A -85,B 0,C 180,E1 -4424.978,E2 -4424.978} C_VEL
LIN {X 0,Y 531.727,Z 322.971,A -85,B 0,C 180,E1 -4427.3,E2 -4427.3} C_VEL
LIN {X 0,Y 532.077,Z 299.564,A -85,B 0,C 180,E1 -4430.085,E2 -4430.085} C_VEL
LIN {X 0,Y 532.518,Z 276.029,A -85,B 0,C 180,E1 -4432.912,E2 -4432.912} C_VEL
LIN {X 0,Y 532.913,Z 249.777,A -85,B 0,C 180,E1 -4436.119,E2 -4436.119} C_VEL
LIN {X 0,Y 530.953,Z 239.536,A -85,B 0,C 180,E1 -4437.479,E2 -4437.479} C_VEL
LIN {X 0,Y 530.937,Z 239.347,A -85,B 0,C 180,E1 -4440.638,E2 -4440.638} C_VEL
LIN {X 0,Y 530.955,Z 239.351,A -85,B 0,C 180,E1 -4443.498,E2 -4443.498} C_VEL
LIN {X 0,Y 530.893,Z 239.35,A -85,B 0,C 180,E1 -4446.145,E2 -4446.145} C_VEL
LIN {X 0,Y 530.926,Z 239.346,A -85,B 0,C 180,E1 -4448.648,E2 -4448.648} C_VEL
LIN {X 0,Y 530.94,Z 239.351,A -85,B 0,C 180,E1 -4451.439,E2 -4451.439} C_VEL
LIN {X 0,Y 530.951,Z 239.343,A -85,B 0,C 180,E1 -4454.549,E2 -4454.549} C_VEL
LIN {X 0,Y 530.903,Z 239.352,A -85,B 0,C 180,E1 -4457.536,E2 -4457.536} C_VEL
LIN {X 0,Y 530.951,Z 239.344,A -85,B 0,C 180,E1 -4460.553,E2 -4460.553} C_VEL
LIN {X 0,Y 530.904,Z 239.352,A -85,B 0,C 180,E1 -4463.437,E2 -4463.437} C_VEL
LIN {X 0,Y 530.922,Z 239.346,A -85,B 0,C 180,E1 -4466.223,E2 -4466.223} C_VEL
LIN {X 0,Y 530.924,Z 239.353,A -85,B 0,C 180,E1 -4468.919,E2 -4468.919} C_VEL
LIN {X 0,Y 530.918,Z 239.348,A -85,B 0,C 180,E1 -4471.54,E2 -4471.54} C_VEL
LIN {X 0,Y 530.917,Z 239.347,A -85,B 0,C 180,E1 -4474.174,E2 -4474.174} C_VEL
LIN {X 0,Y 530.934,Z 239.349,A -85,B 0,C 180,E1 -4476.602,E2 -4476.602} C_VEL
LIN {X 0,Y 530.961,Z 239.347,A -85,B 0,C 180,E1 -4479.061,E2 -4479.061} C_VEL
LIN {X 0,Y 530.952,Z 239.343,A -85,B 0,C 180,E1 -4481.477,E2 -4481.477} C_VEL
LIN {X 0,Y 530.968,Z 239.348,A -85,B 0,C 180,E1 -4484.65,E2 -4484.65} C_VEL
LIN {X 0,Y 531.001,Z 239.336,A -85,B 0,C 180,E1 -4487.774,E2 -4487.774} C_VEL
LIN {X 0,Y 530.949,Z 239.344,A -85,B 0,C 180,E1 -4490.092,E2 -4490.092} C_VEL
LIN {X 0,Y 530.994,Z 239.339,A -85,B 0,C 180,E1 -4493.159,E2 -4493.159} C_VEL
LIN {X 0,Y 530.954,Z 239.342,A -85,B 0,C 180,E1 -4495.445,E2 -4495.445} C_VEL
LIN {X 0,Y 531.109,Z 239.323,A -85,B 0,C 180,E1 -4497.725,E2 -4497.725} C_VEL
LIN {X 0,Y 531.133,Z 239.325,A -85,B 0,C 180,E1 -4500.758,E2 -4500.758} C_VEL
LIN {X 0,Y 531.042,Z 239.333,A -85,B 0,C 180,E1 -4503.035,E2 -4503.035} C_VEL
LIN {X 0,Y 531.025,Z 239.337,A -85,B 0,C 180,E1 -4506.078,E2 -4506.078} C_VEL
LIN {X 0,Y 530.975,Z 239.339,A -85,B 0,C 180,E1 -4509.139,E2 -4509.139} C_VEL
LIN {X 0,Y 530.994,Z 239.345,A -85,B 0,C 180,E1 -4512.226,E2 -4512.226} C_VEL
LIN {X 0,Y 530.969,Z 239.34,A -85,B 0,C 180,E1 -4515.351,E2 -4515.351} C_VEL
LIN {X 0,Y 530.951,Z 239.346,A -85,B 0,C 180,E1 -4518.523,E2 -4518.523} C_VEL
LIN {X 0,Y 530.978,Z 239.339,A -85,B 0,C 180,E1 -4520.939,E2 -4520.939} C_VEL
LIN {X 0,Y 530.941,Z 239.352,A -85,B 0,C 180,E1 -4524.032,E2 -4524.032} C_VEL
LIN {X 0,Y 530.931,Z 239.346,A -85,B 0,C 180,E1 -4526.748,E2 -4526.748} C_VEL
LIN {X 0,Y 530.949,Z 239.343,A -85,B 0,C 180,E1 -4529.325,E2 -4529.325} C_VEL
LIN {X 0,Y 530.943,Z 239.351,A -85,B 0,C 180,E1 -4532.099,E2 -4532.099} C_VEL
LIN {X 0,Y 530.945,Z 239.343,A -85,B 0,C 180,E1 -4534.85,E2 -4534.85} C_VEL
LIN {X 0,Y 530.917,Z 239.35,A -85,B 0,C 180,E1 -4537.512,E2 -4537.512} C_VEL
LIN {X 0,Y 530.898,Z 239.35,A -85,B 0,C 180,E1 -4540.441,E2 -4540.441} C_VEL
LIN {X 0,Y 530.911,Z 239.351,A -85,B 0,C 180,E1 -4543.565,E2 -4543.565} C_VEL
LIN {X 0,Y 530.25,Z 239.433,A -85,B 0,C 180,E1 -4544.199,E2 -4544.199} C_VEL
LIN {X 0,Y 527.413,Z 239.785,A -85,B 0,C 180,E1 -4545.228,E2 -4545.228} C_VEL
LIN {X 0,Y 525.005,Z 240.087,A -85,B 0,C 180,E1 -4546.057,E2 -4546.057} C_VEL
LIN {X 0,Y 523.96,Z 240.213,A -85,B 0,C 180,E1 -4546.697,E2 -4546.697} C_VEL
LIN {X 0,Y 523.869,Z 240.225,A -85,B 0,C 180,E1 -4546.913,E2 -4546.913} C_VEL
LIN {X 0,Y 523.872,Z 240.23,A -85,B 0,C 180,E1 -4549.915,E2 -4549.915} C_VEL
LIN {X 0,Y 523.864,Z 240.225,A -85,B 0,C 180,E1 -4552.866,E2 -4552.866} C_VEL
LIN {X 0,Y 523.899,Z 240.228,A -85,B 0,C 180,E1 -4555.709,E2 -4555.709} C_VEL
LIN {X 0,Y 523.903,Z 240.22,A -85,B 0,C 180,E1 -4558.456,E2 -4558.456} C_VEL
LIN {X 0,Y 523.878,Z 240.227,A -85,B 0,C 180,E1 -4561.123,E2 -4561.123} C_VEL
LIN {X 0,Y 523.877,Z 240.225,A -85,B 0,C 180,E1 -4564.006,E2 -4564.006} C_VEL
LIN {X 0,Y 523.904,Z 240.22,A -85,B 0,C 180,E1 -4566.27,E2 -4566.27} C_VEL
LIN {X 0,Y 523.921,Z 240.219,A -85,B 0,C 180,E1 -4568.766,E2 -4568.766} C_VEL
LIN {X 0,Y 523.916,Z 240.226,A -85,B 0,C 180,E1 -4571.22,E2 -4571.22} C_VEL
LIN {X 0,Y 523.887,Z 240.226,A -85,B 0,C 180,E1 -4573.638,E2 -4573.638} C_VEL
LIN {X 0,Y 523.898,Z 240.221,A -85,B 0,C 180,E1 -4576.028,E2 -4576.028} C_VEL
LIN {X 0,Y 523.971,Z 240.213,A -85,B 0,C 180,E1 -4578.394,E2 -4578.394} C_VEL
LIN {X 0,Y 523.937,Z 240.224,A -85,B 0,C 180,E1 -4581.515,E2 -4581.515} C_VEL
LIN {X 0,Y 524,Z 240.372,A -85,B 0,C 180,E1 -4583.024,E2 -4583.024} C_VEL
LIN {X 0,Y 524.172,Z 241.187,A -85,B 0,C 180,E1 -4583.142,E2 -4583.142} C_VEL
LIN {X 0,Y 526.012,Z 247.209,A -85,B 0,C 180,E1 -4583.3,E2 -4583.3} C_VEL
LIN {X 0,Y 525.634,Z 328.82,A -85,B 0,C 180,E1 -4584.438,E2 -4584.438} C_VEL
LIN {X 0,Y 525.516,Z 341.905,A -85,B 0,C 180,E1 -4584.773,E2 -4584.773} C_VEL
LIN {X 0,Y 525.351,Z 354.428,A -85,B 0,C 180,E1 -4585.252,E2 -4585.252} C_VEL
LIN {X 0,Y 525.122,Z 366.386,A -85,B 0,C 180,E1 -4585.875,E2 -4585.875} C_VEL
LIN {X 0,Y 524.867,Z 377.704,A -85,B 0,C 180,E1 -4586.642,E2 -4586.642} C_VEL
LIN {X 0,Y 524.581,Z 387.901,A -85,B 0,C 180,E1 -4587.505,E2 -4587.505} C_VEL
LIN {X 0,Y 524.357,Z 397.097,A -85,B 0,C 180,E1 -4588.464,E2 -4588.464} C_VEL
LIN {X 0,Y 524.099,Z 405.972,A -85,B 0,C 180,E1 -4589.616,E2 -4589.616} C_VEL
LIN {X 0,Y 523.898,Z 413.134,A -85,B 0,C 180,E1 -4590.769,E2 -4590.769} C_VEL
LIN {X 0,Y 523.669,Z 418.901,A -85,B 0,C 180,E1 -4591.923,E2 -4591.923} C_VEL
LIN {X 0,Y 523.613,Z 423.438,A -85,B 0,C 180,E1 -4593.078,E2 -4593.078} C_VEL
LIN {X 0,Y 523.576,Z 425.868,A -85,B 0,C 180,E1 -4593.849,E2 -4593.849} C_VEL
LIN {X 0,Y 523.572,Z 427.834,A -85,B 0,C 180,E1 -4594.62,E2 -4594.62} C_VEL
LIN {X 0,Y 523.507,Z 430.58,A -85,B 0,C 180,E1 -4596.166,E2 -4596.166} C_VEL
LIN {X 0,Y 523.53,Z 431.317,A -85,B 0,C 180,E1 -4596.939,E2 -4596.939} C_VEL
LIN {X 0,Y 523.466,Z 431.659,A -85,B 0,C 180,E1 -4598.493,E2 -4598.493} C_VEL
LIN {X 0,Y 523.458,Z 431.258,A -85,B 0,C 180,E1 -4599.272,E2 -4599.272} C_VEL
LIN {X 0,Y 523.449,Z 430.421,A -85,B 0,C 180,E1 -4600.052,E2 -4600.052} C_VEL
LIN {X 0,Y 523.566,Z 427.787,A -85,B 0,C 180,E1 -4601.503,E2 -4601.503} C_VEL
LIN {X 0,Y 523.63,Z 424.203,A -85,B 0,C 180,E1 -4602.795,E2 -4602.795} C_VEL
LIN {X 0,Y 523.697,Z 419.767,A -85,B 0,C 180,E1 -4603.979,E2 -4603.979} C_VEL
LIN {X 0,Y 523.903,Z 412.96,A -85,B 0,C 180,E1 -4605.363,E2 -4605.363} C_VEL
LIN {X 0,Y 524.112,Z 405.483,A -85,B 0,C 180,E1 -4606.556,E2 -4606.556} C_VEL
LIN {X 0,Y 524.332,Z 397.12,A -85,B 0,C 180,E1 -4607.633,E2 -4607.633} C_VEL
LIN {X 0,Y 524.633,Z 387.252,A -85,B 0,C 180,E1 -4608.653,E2 -4608.653} C_VEL
LIN {X 0,Y 524.884,Z 376.385,A -85,B 0,C 180,E1 -4609.557,E2 -4609.557} C_VEL
LIN {X 0,Y 525.183,Z 365.748,A -85,B 0,C 180,E1 -4610.259,E2 -4610.259} C_VEL
LIN {X 0,Y 525.39,Z 353.231,A -85,B 0,C 180,E1 -4610.894,E2 -4610.894} C_VEL
LIN {X 0,Y 525.559,Z 340.344,A -85,B 0,C 180,E1 -4611.37,E2 -4611.37} C_VEL
LIN {X 0,Y 525.71,Z 327.685,A -85,B 0,C 180,E1 -4611.673,E2 -4611.673} C_VEL
LIN {X 0,Y 525.919,Z 246.448,A -85,B 0,C 180,E1 -4612.805,E2 -4612.805} C_VEL
LIN {X 0,Y 524.094,Z 241.039,A -85,B 0,C 180,E1 -4612.965,E2 -4612.965} C_VEL
LIN {X 0,Y 523.93,Z 240.315,A -85,B 0,C 180,E1 -4613.101,E2 -4613.101} C_VEL
LIN {X 0,Y 523.912,Z 240.224,A -85,B 0,C 180,E1 -4616.002,E2 -4616.002} C_VEL
LIN {X 0,Y 523.927,Z 240.226,A -85,B 0,C 180,E1 -4618.875,E2 -4618.875} C_VEL
LIN {X 0,Y 523.92,Z 240.215,A -85,B 0,C 180,E1 -4621.544,E2 -4621.544} C_VEL
LIN {X 0,Y 523.914,Z 240.224,A -85,B 0,C 180,E1 -4624.291,E2 -4624.291} C_VEL
LIN {X 0,Y 523.883,Z 240.219,A -85,B 0,C 180,E1 -4627.134,E2 -4627.134} C_VEL
LIN {X 0,Y 523.912,Z 240.223,A -85,B 0,C 180,E1 -4630.126,E2 -4630.126} C_VEL
LIN {X 0,Y 523.888,Z 240.225,A -85,B 0,C 180,E1 -4633.169,E2 -4633.169} C_VEL
LIN {X 0,Y 523.916,Z 240.219,A -85,B 0,C 180,E1 -4635.769,E2 -4635.769} C_VEL
LIN {X 0,Y 523.894,Z 240.225,A -85,B 0,C 180,E1 -4638.903,E2 -4638.903} C_VEL
LIN {X 0,Y 523.898,Z 240.221,A -85,B 0,C 180,E1 -4641.896,E2 -4641.896} C_VEL
LIN {X 0,Y 523.912,Z 240.222,A -85,B 0,C 180,E1 -4644.912,E2 -4644.912} C_VEL
LIN {X 0,Y 523.93,Z 240.218,A -85,B 0,C 180,E1 -4647.679,E2 -4647.679} C_VEL
LIN {X 0,Y 523.948,Z 240.214,A -85,B 0,C 180,E1 -4650.676,E2 -4650.676} C_VEL
LIN {X 0,Y 523.915,Z 240.226,A -85,B 0,C 180,E1 -4653.994,E2 -4653.994} C_VEL
LIN {X 0,Y 523.904,Z 240.219,A -85,B 0,C 180,E1 -4656.269,E2 -4656.269} C_VEL
LIN {X 0,Y 523.938,Z 240.208,A -85,B 0,C 180,E1 -4658.766,E2 -4658.766} C_VEL
LIN {X 0,Y 523.929,Z 240.216,A -85,B 0,C 180,E1 -4661.22,E2 -4661.22} C_VEL
LIN {X 0,Y 523.908,Z 240.224,A -85,B 0,C 180,E1 -4663.638,E2 -4663.638} C_VEL
LIN {X 0,Y 523.917,Z 240.225,A -85,B 0,C 180,E1 -4666.027,E2 -4666.027} C_VEL
LIN {X 0,Y 524.006,Z 240.21,A -85,B 0,C 180,E1 -4668.394,E2 -4668.394} C_VEL
LIN {X 0,Y 523.945,Z 240.216,A -85,B 0,C 180,E1 -4671.515,E2 -4671.515} C_VEL
LIN {X 0,Y 524.027,Z 240.204,A -85,B 0,C 180,E1 -4674.613,E2 -4674.613} C_VEL
LIN {X 0,Y 524.092,Z 240.203,A -85,B 0,C 180,E1 -4677.694,E2 -4677.694} C_VEL
LIN {X 0,Y 524.083,Z 240.201,A -85,B 0,C 180,E1 -4680,E2 -4680} C_VEL
LIN {X 0,Y 524.024,Z 240.205,A -85,B 0,C 180,E1 -4683.075,E2 -4683.075} C_VEL
LIN {X 0,Y 523.987,Z 240.21,A -85,B 0,C 180,E1 -4686.16,E2 -4686.16} C_VEL
LIN {X 0,Y 523.966,Z 240.216,A -85,B 0,C 180,E1 -4689.262,E2 -4689.262} C_VEL
LIN {X 0,Y 523.986,Z 240.212,A -85,B 0,C 180,E1 -4691.735,E2 -4691.735} C_VEL
LIN {X 0,Y 523.974,Z 240.215,A -85,B 0,C 180,E1 -4695.048,E2 -4695.048} C_VEL
LIN {X 0,Y 523.935,Z 240.216,A -85,B 0,C 180,E1 -4697.97,E2 -4697.97} C_VEL
LIN {X 0,Y 523.943,Z 240.216,A -85,B 0,C 180,E1 -4700.411,E2 -4700.411} C_VEL
LIN {X 0,Y 523.898,Z 240.224,A -85,B 0,C 180,E1 -4702.894,E2 -4702.894} C_VEL
LIN {X 0,Y 523.888,Z 240.225,A -85,B 0,C 180,E1 -4705.422,E2 -4705.422} C_VEL
LIN {X 0,Y 523.889,Z 240.217,A -85,B 0,C 180,E1 -4708.004,E2 -4708.004} C_VEL
LIN {X 0,Y 523.892,Z 240.228,A -85,B 0,C 180,E1 -4710.846,E2 -4710.846} C_VEL
LIN {X 0,Y 523.92,Z 240.214,A -85,B 0,C 180,E1 -4713.729,E2 -4713.729} C_VEL
LIN {X 0,Y 523.861,Z 240.228,A -85,B 0,C 180,E1 -4716.396,E2 -4716.396} C_VEL
LIN {X 0,Y 523.904,Z 240.225,A -85,B 0,C 180,E1 -4719.086,E2 -4719.086} C_VEL
LIN {X 0,Y 523.886,Z 240.224,A -85,B 0,C 180,E1 -4722.126,E2 -4722.126} C_VEL
LIN {X 0,Y 523.926,Z 240.22,A -85,B 0,C 180,E1 -4725.312,E2 -4725.312} C_VEL
LIN {X 0,Y 523.905,Z 240.228,A -85,B 0,C 180,E1 -4728.696,E2 -4728.696} C_VEL
LIN {X 0,Y 523.873,Z 240.223,A -85,B 0,C 180,E1 -4731.895,E2 -4731.895} C_VEL
LIN {X 0,Y 523.91,Z 240.221,A -85,B 0,C 180,E1 -4734.914,E2 -4734.914} C_VEL
LIN {X 0,Y 523.898,Z 240.221,A -85,B 0,C 180,E1 -4737.686,E2 -4737.686} C_VEL
LIN {X 0,Y 523.864,Z 240.23,A -85,B 0,C 180,E1 -4740.24,E2 -4740.24} C_VEL
LIN {X 0,Y 523.917,Z 240.433,A -85,B 0,C 180,E1 -4742.379,E2 -4742.379} C_VEL
LIN {X 0,Y 525.758,Z 249.255,A -85,B 0,C 180,E1 -4743.588,E2 -4743.588} C_VEL
LIN {X 0,Y 525.769,Z 259.552,A -85,B 0,C 180,E1 -4744.881,E2 -4744.881} C_VEL
LIN {X 0,Y 525.331,Z 283.605,A -85,B 0,C 180,E1 -4747.833,E2 -4747.833} C_VEL
LIN {X 0,Y 524.893,Z 306.868,A -85,B 0,C 180,E1 -4750.647,E2 -4750.647} C_VEL
LIN {X 0,Y 524.585,Z 328.643,A -85,B 0,C 180,E1 -4753.259,E2 -4753.259} C_VEL
LIN {X 0,Y 524.419,Z 341.814,A -85,B 0,C 180,E1 -4754.808,E2 -4754.808} C_VEL
LIN {X 0,Y 525.904,Z 356.821,A -85,B 0,C 180,E1 -4755.075,E2 -4755.075} C_VEL
LIN {X 0,Y 525.439,Z 451.885,A -85,B 0,C 180,E1 -4756.389,E2 -4756.389} C_VEL
LIN {X 0,Y 525.185,Z 465.253,A -85,B 0,C 180,E1 -4756.727,E2 -4756.727} C_VEL
LIN {X 0,Y 524.958,Z 478.659,A -85,B 0,C 180,E1 -4757.238,E2 -4757.238} C_VEL
LIN {X 0,Y 524.675,Z 490.914,A -85,B 0,C 180,E1 -4757.881,E2 -4757.881} C_VEL
LIN {X 0,Y 524.353,Z 502.973,A -85,B 0,C 180,E1 -4758.696,E2 -4758.696} C_VEL
LIN {X 0,Y 524.092,Z 513.313,A -85,B 0,C 180,E1 -4759.57,E2 -4759.57} C_VEL
LIN {X 0,Y 523.881,Z 522.633,A -85,B 0,C 180,E1 -4760.541,E2 -4760.541} C_VEL
LIN {X 0,Y 523.704,Z 531.728,A -85,B 0,C 180,E1 -4761.705,E2 -4761.705} C_VEL
LIN {X 0,Y 523.572,Z 539.062,A -85,B 0,C 180,E1 -4762.867,E2 -4762.867} C_VEL
